(* CODESYS project almacen.project
   Version: 0.0.0.0
   Title: prueba_v2
   Author: Sara

Project tree, tasks and I/O mapping:
  MyController : TM241CE24R, Schneider Electric, order no. TM241CE24R, version 5.0.8.2
    application Application
      libraries: VisuElemBase, * (System); VisuDialogs, * (System)
      task MAST (cyclic, interval 10 ms, priority 15, watchdog 100 ms x 1) calls Main
      task VISU_TASK (cyclic, interval 100 ms, priority 31) calls VisuElems.Visu_Prg
      global variables GVL
      program Main [ST]
      program RecogidaPieza [ST]: Inicio_PiezaEntrada, PiezaDetectada
      program PosicionRobot [ST]
      program TrasladoPieza [ST]: Inicio_TrasladoPieza
      program ExtraerPieza [ST]: Inicio_ExtraerPieza
      program SalidaPieza [ST]: Inicio_SalidaPieza
      program Seguridad [ST]
      program MovimientoRobot [ST]: Inicio_MovimientoRobot, Fin_MovRobot
      program Funcionamiento [ST]: Carga, Descarga, NoAlmacena, CargaDescarga, CD_NoCarga, CD_Carga, CD_Descarga, CD_NoDescarga, ConfirmaCarga
      program Mando [ST]: Inicializar, Automatico, Manual, ParadaSolicitada
      program Acciones [ST]
      program Inicializacion [ST]
      program GestionPiezas [ST]
      program MarchaVSO [ST]: Recoger, Trasladar, Extraer, Salir, Finalizar
      program Comunicacion [CFC]
      program EntradasSalidas [ST]
      text list Pantallas_Lista
      program Control [ST]
      text list Funcionamiento_Lista
      text list Descarga_Lista
      text list DescargaColor_Lista
      program Test [ST]: Subir, Bajar, Estirar, Recoger, Abrir, Cerrar
      text list Test_Lista
      text list Carga_Lista
      Etapas/
        data type Etapas_RecogidaPieza
        data type Etapas_TrasladoPieza
        data type Etapas_ExtraerPieza
        data type Etapas_SalidaPieza
        data type Etapas_Seguridad
        data type Etapas_MovimientoRobot
        data type Etapas_Funcionamiento
        data type Etapas_Mando
        data type Etapas_Inicializacion
        data type Etapas_MarchaVSO
        data type Etapas_Test
      visualisation Pantalla
    DI : Digital Inputs, Schneider Electric, version 5.0.8.2
        input  iwDI_IW0 : WORD  // IW0
        input  ibDI_IB1 : BYTE  // IB1
    DQ : Digital Outputs, Schneider Electric, version 5.0.8.2
        output qwDQ_QW0 : WORD  // QW0
        output qbDQ_QB1 : BYTE  // QB1
    Counters : Counters, Schneider Electric, version 5.0.8.2
    Pulse_Generators : Pulse Generators, Schneider Electric, version 5.0.8.2
    Cartridge_1 : Cartridge, Schneider Electric, version 5.0.8.2
    IO_Bus : IO bus - TM3, Schneider Electric, version 5.0.8.2
    COM_Bus : COM bus, Schneider Electric, version 5.0.8.2
    Ethernet_1 : Ethernet Network, Schneider Electric, version 5.0.8.2
        settings: IPAddress = [10, 11, 164, 211]; SubnetMask = [255, 255, 252, 0]; WebServer = TRUE; FTP Server = TRUE; SoMachine Protocol = TRUE; Modbus Server = TRUE; NetManage Protocol = TRUE; SNMP protocol = TRUE; Enable Routing = FALSE; WebVisu protocol = TRUE; DHCP Server Active = TRUE
    Serial_Line_1 : Serial line, Schneider Electric, version 5.0.8.2
      Machine_Expert_Network_Manager : Machine Expert-Network Manager, Schneider Electric, version 4.0.0.3
    Serial_Line_2 : Serial line, Schneider Electric, version 5.0.8.2
      Modbus_Manager : Modbus Manager, Schneider Electric, version 4.0.0.3
  libraries: VisuSymbols, 3.5.10.0 (System)
  text list GlobalTextList
*)

// MyController/Application/Etapas/Etapas_RecogidaPieza
{attribute 'qualified_only'}
{attribute 'strict'}
TYPE Etapas_RecogidaPieza :
(
	EInicial, RecogerCilindro1, MoverRobot, AccionarCilindro, DetectarPieza,
	Espera, BajarRobot, CerrarPinza, SubirRobot, RecogerCilindro2 
);
END_TYPE

// MyController/Application/Etapas/Etapas_TrasladoPieza
{attribute 'qualified_only'}
{attribute 'strict'}
TYPE Etapas_TrasladoPieza :
(
	EInicial, MoverRobot, AccionarCilindro, BajarRobot, AbrirPinza, SubirRobot, 
	RecogerCilindro, Fin
);
END_TYPE

// MyController/Application/Etapas/Etapas_ExtraerPieza
{attribute 'qualified_only'}
{attribute 'strict'}
TYPE Etapas_ExtraerPieza :
(
	EInicial, RecogerCilindro1, MoverRobot, AccionarCilindro, BajarRobot, CerrarPinza,
	SubirRobot, RecogerCilindro2, Espera
);
END_TYPE

// MyController/Application/Etapas/Etapas_SalidaPieza
{attribute 'qualified_only'}
{attribute 'strict'}
TYPE Etapas_SalidaPieza :
(
	EInicial, MoverRobot, AccionarCilindro, AbrirPinza, SubirRobot, RecogerCilindro, Fin
);
END_TYPE

// MyController/Application/Etapas/Etapas_Seguridad
{attribute 'qualified_only'}
{attribute 'strict'}
TYPE Etapas_Seguridad :
(
	Normal, D1, Rearme
);
END_TYPE

// MyController/Application/Etapas/Etapas_MovimientoRobot
{attribute 'qualified_only'}
{attribute 'strict'}
TYPE Etapas_MovimientoRobot :
(
	EInicial, EnvioVertical, MovVertical, EnvioHorizontal, MovHorizontal, Fin
);
END_TYPE

// MyController/Application/Etapas/Etapas_Funcionamiento
{attribute 'qualified_only'}
{attribute 'strict'}
TYPE Etapas_Funcionamiento :
(
	EInicial, Modo, RecogePieza1, SalidaPieza, RecogePieza2, TrasladoPieza, Espera,
	ExtraePieza, EsperaCD_Carga, EsperaCD_Descarga, SalidaPieza2, Fin
);
END_TYPE

// MyController/Application/Etapas/Etapas_Mando
{attribute 'qualified_only'}
{attribute 'strict'}
TYPE Etapas_Mando :
(
	A1, A2, A6, F1, F4, F6
);
END_TYPE

// MyController/Application/Etapas/Etapas_Inicializacion
{attribute 'qualified_only'}
{attribute 'strict'}
TYPE Etapas_Inicializacion :
(
	EInicial, Espera, MoverRobot, Fin
);
END_TYPE

// MyController/Application/Etapas/Etapas_MarchaVSO
{attribute 'qualified_only'}
{attribute 'strict'}
TYPE Etapas_MarchaVSO :
(
	EInicial, Funcionamiento, RecogePieza, TrasladoPieza, ExtraePieza, SalidaPieza, Espera, Fin
);
END_TYPE

// MyController/Application/Etapas/Etapas_Test
{attribute 'qualified_only'}
{attribute 'strict'}
TYPE Etapas_Test :
(
	EInicial, Espera, Funcionamiento, MoverRobot, SubirRobot, BajarRobot, AccionarCilindro, RecogerCilindro,
	AbrirPinza, CerrarPinza, Fin
);
END_TYPE

// MyController/Application/GVL
{attribute 'qualified_only'}
VAR_GLOBAL
	// Selector (AUTO=0, MAN=1)
	IN_Aut_Man: BOOL;
	// Final de carrera activado con el cilindro recogido
	IN_FC_CilindroAtras: BOOL;
	// Final de carrera activado con el cilindro accionado
	IN_FC_CilindroDelante: BOOL;
	// Final del movimiento horizontal del robot detectado
	IN_Fin_EjeHorizontal: BOOL;
	// Final del movimiento vertical del robot detectado
	IN_Fin_EjeVertical: BOOL;
	// Detector de pieza negra
	IN_PiezaNegra: BOOL;
	// Detector de pieza roja
	IN_PiezaRoja: BOOL;
	// Detector de pieza plateada
	IN_PiezaPlateada: BOOL;
	// Pulsador Reset
	IN_Reset: BOOL;
	// Seta de emergencia
	IN_Seta_Emergencia: BOOL;
	// Pulsador Start
	IN_Start: BOOL;
	// Pulsador Stop
	IN_Stop: BOOL;
	// Bit de posición 0
	OUT_Bit_Posicion0: BOOL;
	// Bit de posición 1
	OUT_Bit_Posicion1: BOOL;
	// Bit de posición 2
	OUT_Bit_Posicion2: BOOL;
	// Accionar el cilindro
	OUT_Cilindro: BOOL;
	// Inicio del movimiento horizontal del robot
	OUT_EjeHorizontal: BOOL;
	// Inicio del movimiento vertical del robot
	OUT_EjeVertical: BOOL;
	// Piloto Q1
	OUT_Piloto_Q1: BOOL;
	// Piloto Q2
	OUT_Piloto_Q2: BOOL;
	// Piloto Reset
	OUT_Piloto_Reset: BOOL;
	// Piloto Start
	OUT_Piloto_Start: BOOL;
	// Accionar la pinza
	OUT_Pinza: BOOL;
	// Bit que indica que hay una pieza en la entrada 
	// (escrito por la estación de procesado)
	BIT_PiezaEntrada: BOOL;
	// Bit que indica que se ha recogido la pieza de la entrada
	// (leído por la estación de procesado)
	BIT_PiezaRecogida: BOOL;
END_VAR

// MyController/Application/Main
PROGRAM Main
VAR
	VSO_Recoger: BOOL;
	VSO_Extraer: BOOL;
	VSO_Salir: BOOL;
	VSO_Trasladar: BOOL;
	VSO_Nada: BOOL;
	VSO_ColorDescarga: INT;
END_VAR

Comunicacion();
EntradasSalidas();
Funcionamiento();
Mando();
Seguridad();
RecogidaPieza();
TrasladoPieza();
ExtraerPieza();
SalidaPieza();
Inicializacion();
Acciones();
MovimientoRobot();
PosicionRobot();
GestionPiezas();
MarchaVSO();
Control();
Test();

END_PROGRAM

// MyController/Application/Comunicacion
PROGRAM Comunicacion
VAR
	FB_ADDM: ADDM;
	FB_READ_VAR: READ_VAR;
	FB_WRITE_VAR: WRITE_VAR;
	DataRead: ARRAY [0..0] OF WORD;
	DataWrite: ARRAY [0..0] OF WORD;
	Direccion: ADDRESS;
	addm_exe: BOOL;
	Q_TIMER0:BOOL;
	TON_0: TON;
	CTU0: CTU;
	SR: SR;
END_VAR

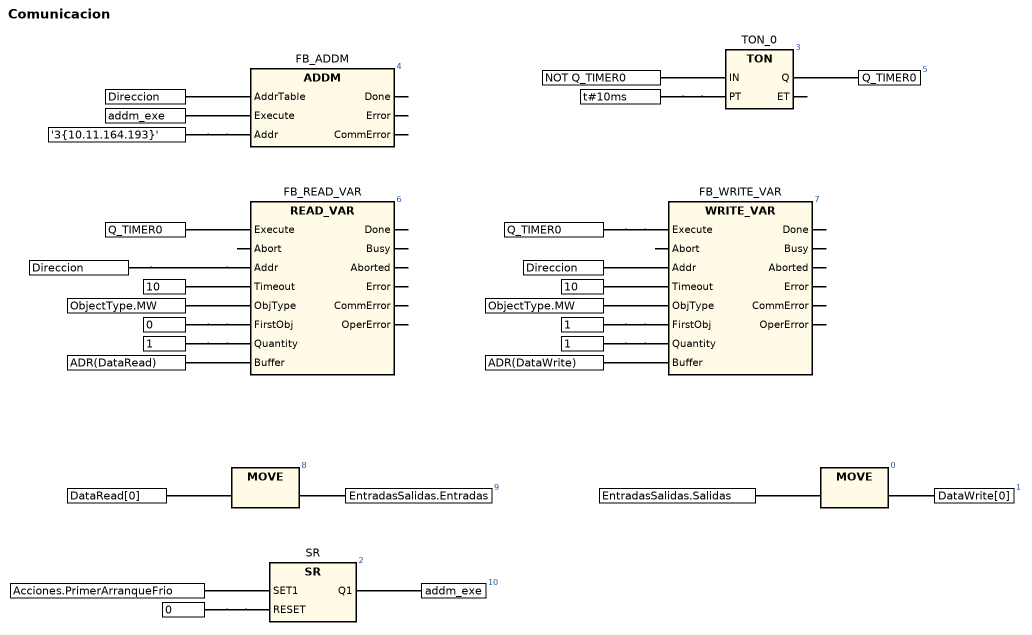
DataWrite[0] := EntradasSalidas.Salidas;
SR(SET1 := Acciones.PrimerArranqueFrio, RESET := 0);
TON_0(IN := NOT Q_TIMER0, PT := t#10ms); // TON
FB_ADDM(AddrTable := Direccion, Execute := addm_exe, Addr := '3{10.11.164.193}'); // ADDM
Q_TIMER0 := TON_0.Q;
FB_READ_VAR(
    Execute := Q_TIMER0,
    Addr := Direccion,
    Timeout := 10,
    ObjType := ObjectType.MW,
    FirstObj := 0,
    Quantity := 1,
    Buffer := ADR(DataRead)); // READ_VAR
FB_WRITE_VAR(
    Execute := Q_TIMER0,
    Addr := Direccion,
    Timeout := 10,
    ObjType := ObjectType.MW,
    FirstObj := 1,
    Quantity := 1,
    Buffer := ADR(DataWrite)); // WRITE_VAR
EntradasSalidas.Entradas := DataRead[0];
addm_exe := SR.Q1;

END_PROGRAM

// MyController/Application/EntradasSalidas
PROGRAM EntradasSalidas
VAR_INPUT
	Entradas: WORD;
END_VAR
VAR
	Salidas: WORD;
END_VAR

(*ENTRADAS*)
GVL.IN_Start := Entradas.0;
GVL.IN_Stop := Entradas.1;
GVL.IN_Reset := Entradas.3;
GVL.IN_Seta_Emergencia := Entradas.5;
GVL.IN_FC_CilindroAtras := Entradas.8;
GVL.IN_FC_CilindroDelante := Entradas.9;
GVL.IN_PiezaNegra := Entradas.10;
GVL.IN_PiezaRoja := Entradas.11;
GVL.IN_PiezaPlateada := Entradas.12;
GVL.IN_Fin_EjeVertical := Entradas.13;
GVL.IN_Fin_EjeHorizontal := Entradas.14;
GVL.BIT_PiezaEntrada := Entradas.15;

(*SALIDAS*)
Salidas.0 := GVL.OUT_Piloto_Start;
Salidas.1 := GVL.OUT_Piloto_Reset;
Salidas.2 := GVL.OUT_Piloto_Q1;
Salidas.3 := GVL.OUT_Piloto_Q2;
Salidas.4 := GVL.OUT_Cilindro;
Salidas.5 := GVL.OUT_Pinza;
Salidas.6 := GVL.OUT_Bit_Posicion0;
Salidas.7 := GVL.OUT_Bit_Posicion1;
Salidas.8 := GVL.OUT_Bit_Posicion2;
Salidas.9 := GVL.OUT_EjeVertical;
Salidas.10 := GVL.OUT_EjeHorizontal;
Salidas.11 := GVL.BIT_PiezaRecogida;

END_PROGRAM

// MyController/Application/Acciones
PROGRAM Acciones
VAR
	SET_Cilindro: BOOL;
	RESET_Cilindro: BOOL;
	SET_Pinza: BOOL;
	RESET_Pinza: BOOL;
	BLINK: BLINK;
	PrimerArranqueFrio: BOOL;
	SR_1: SR;
	SR_3: SR;
	SR_4: SR;
	Parpadeo: BOOL;
	TON: ton;
	Tiempo_350ms: BOOL;
	EntradaTON350ms: BOOL;
	TON_3: TON;
	EntradaTON500ms: BOOL;
	Tiempo_500ms: BOOL;
	TON_2: TON;
	EntradaTON1s: BOOL;
	Tiempo_1s: BOOL;
END_VAR

(*PARADA DE EMERGENCIA*)
IF Seguridad.Estado = Etapas_Seguridad.D1 THEN
	RecogidaPieza.Estado := Etapas_RecogidaPieza.EInicial;
	TrasladoPieza.Estado := Etapas_TrasladoPieza.EInicial;
	ExtraerPieza.Estado := Etapas_ExtraerPieza.EInicial;
	SalidaPieza.Estado := Etapas_SalidaPieza.EInicial;
	MovimientoRobot.Estado := Etapas_MovimientoRobot.EInicial;
	Mando.Estado := Etapas_Mando.A1;
	Funcionamiento.Estado := Etapas_Funcionamiento.EInicial;
	Inicializacion.Estado := Etapas_Inicializacion.EInicial;
	MarchaVSO.Estado := Etapas_MarchaVSO.EInicial;
END_IF

(*REARME*)
IF Seguridad.Estado = Etapas_Seguridad.Rearme THEN
	Mando.Estado := Etapas_Mando.A6;
END_IF


(*GUARDAR FECHA Y COLOR TEMPORAL PARA LA GESTIÓN DE PIEZAS*)
IF RecogidaPieza.Estado = Etapas_RecogidaPieza.DetectarPieza THEN
	IF GVL.IN_PiezaNegra THEN
		RecogidaPieza.ColorPieza := 1;
		RecogidaPieza.Fecha := getRTC();
	ELSIF GVL.IN_PiezaPlateada THEN
		RecogidaPieza.ColorPieza := 2;
		RecogidaPieza.Fecha := getRTC();
	ELSIF GVL.IN_PiezaRoja THEN
		RecogidaPieza.ColorPieza := 3;
		RecogidaPieza.Fecha := getRTC();
	END_IF 
END_IF


(*ACCIONAMIENTO DEL CILINDRO*)
IF RecogidaPieza.Estado = Etapas_RecogidaPieza.AccionarCilindro OR TrasladoPieza.Estado = Etapas_TrasladoPieza.AccionarCilindro OR 
	ExtraerPieza.Estado = Etapas_ExtraerPieza.AccionarCilindro OR SalidaPieza.Estado = Etapas_SalidaPieza.AccionarCilindro OR
	Test.Estado = Etapas_Test.AccionarCilindro THEN
	  SET_Cilindro := 1;
ELSE			
	  SET_Cilindro := 0;	
END_IF

(*RECOGIDA DEL CILINDRO*)
IF RecogidaPieza.Estado = Etapas_RecogidaPieza.RecogerCilindro1 OR RecogidaPieza.Estado = Etapas_RecogidaPieza.RecogerCilindro2 OR
	TrasladoPieza.Estado = Etapas_TrasladoPieza.RecogerCilindro OR ExtraerPieza.Estado = Etapas_ExtraerPieza.RecogerCilindro1 OR
	ExtraerPieza.Estado = Etapas_ExtraerPieza.RecogerCilindro2 OR SalidaPieza.Estado = Etapas_SalidaPieza.RecogerCilindro 
	OR Inicializacion.Estado = Etapas_Inicializacion.Espera OR Seguridad.Estado = Etapas_Seguridad.D1 OR
	Test.Estado = Etapas_Test.RecogerCilindro THEN
	  RESET_Cilindro := 1;
ELSE			
	  RESET_Cilindro := 0;	
END_IF

(*ABRIR LA PINZA*)
IF TrasladoPieza.Estado = Etapas_TrasladoPieza.AbrirPinza OR SalidaPieza.Estado = Etapas_SalidaPieza.AbrirPinza OR
	Inicializacion.Estado = Etapas_Inicializacion.Espera OR Seguridad.Estado = Etapas_Seguridad.D1 OR 
	Test.Estado = Etapas_Test.AbrirPinza THEN
	  RESET_Pinza := 1;
ELSE			
	  RESET_Pinza := 0;	
END_IF

(*CERRAR LA PINZA*)
IF RecogidaPieza.Estado = Etapas_RecogidaPieza.CerrarPinza OR  ExtraerPieza.Estado = Etapas_ExtraerPieza.CerrarPinza OR
	Test.Estado = Etapas_Test.CerrarPinza THEN
	  SET_Pinza:= 1;
ELSE			
	  SET_Pinza := 0;	
END_IF


(*ARRANQUE FRÍO*)
PrimerArranqueFrio := IsFirstMastColdCycle();
SR_1(SET1:= PrimerArranqueFrio, RESET:= Mando.Estado = Etapas_Mando.A6, Q1=> Mando.ArranqueFrio);


(*TEMPORIZADOR 350ms*)
IF MovimientoRobot.Estado = Etapas_MovimientoRobot.EnvioVertical OR MovimientoRobot.Estado = Etapas_MovimientoRobot.EnvioHorizontal  THEN
		EntradaTON350ms := 1;
ELSE
		EntradaTON350ms := 0;
END_IF
TON(IN:= EntradaTON350ms, PT:= T#350MS, Q=> Tiempo_350ms);

(*TEMPORIZADOR 1s*)
IF TrasladoPieza.Estado = Etapas_TrasladoPieza.MoverRobot THEN
	EntradaTON1s := 1;
ELSE
	EntradaTON1s := 0;
END_IF
TON_2(IN:= EntradaTON1s, PT:= T#1S, Q=> Tiempo_1s);

(*TEMPORIZADOR 500ms*)
IF RecogidaPieza.Estado = Etapas_RecogidaPieza.DetectarPieza  OR MovimientoRobot.Estado = Etapas_MovimientoRobot.MovVertical OR 
	MovimientoRobot.Estado = Etapas_MovimientoRobot.MovHorizontal OR RecogidaPieza.Estado = Etapas_RecogidaPieza.Espera THEN
	EntradaTON500ms := 1;
ELSE
	EntradaTON500ms := 0;
END_IF
TON_3(IN:= EntradaTON500ms, PT:= T#500MS, Q=> Tiempo_500ms);

BLINK(ENABLE:= TRUE, TIMELOW:= T#500MS, TIMEHIGH:= T#500MS, OUT=> Parpadeo);


(*SALIDAS*)
(*BIT_PIEZARECOGIDA*)
GVL.BIT_PiezaRecogida := RecogidaPieza.Estado = Etapas_RecogidaPieza.Espera;

(*OUT_CILINDRO*)
SR_3(SET1:= SET_Cilindro , RESET:= RESET_Cilindro, Q1=> GVL.OUT_Cilindro );

(*OUT_PINZA*)
SR_4(SET1:= SET_Pinza , RESET:= RESET_Pinza, Q1=> GVL.OUT_Pinza );

(*OUT_BIT_POSICION*)
CASE PosicionRobot.EnviarCoordenadas OF
	0: GVL.OUT_Bit_Posicion2:=0; GVL.OUT_Bit_Posicion1:=0; GVL.OUT_Bit_Posicion0:=0;
	1: GVL.OUT_Bit_Posicion2:=0; GVL.OUT_Bit_Posicion1:=0; GVL.OUT_Bit_Posicion0:=1;
	2: GVL.OUT_Bit_Posicion2:=0; GVL.OUT_Bit_Posicion1:=1; GVL.OUT_Bit_Posicion0:=0;
	3: GVL.OUT_Bit_Posicion2:=0; GVL.OUT_Bit_Posicion1:=1; GVL.OUT_Bit_Posicion0:=1;
	4: GVL.OUT_Bit_Posicion2:=1; GVL.OUT_Bit_Posicion1:=0; GVL.OUT_Bit_Posicion0:=0;
	5: GVL.OUT_Bit_Posicion2:=1; GVL.OUT_Bit_Posicion1:=0; GVL.OUT_Bit_Posicion0:=1;
	6: GVL.OUT_Bit_Posicion2:=1; GVL.OUT_Bit_Posicion1:=1; GVL.OUT_Bit_Posicion0:=0;
	7: GVL.OUT_Bit_Posicion2:=1; GVL.OUT_Bit_Posicion1:=1; GVL.OUT_Bit_Posicion0:=1;
END_CASE

(*OUT_EJEVERTICAL*)
IF MovimientoRobot.Estado = Etapas_MovimientoRobot.MovVertical THEN
	GVL.OUT_EjeVertical := 1;
ELSE 
	GVL.OUT_EjeVertical := 0;
END_IF

(*OUT_EJEHORIZONTAL*)
IF MovimientoRobot.Estado = Etapas_MovimientoRobot.MovHorizontal THEN
	GVL.OUT_EjeHorizontal := 1;
ELSE
	GVL.OUT_EjeHorizontal := 0;
END_IF

(*OUT_PILOTO_Q1*)
(*Se enciende de forma continua cuando la estación está EN FUNCIONAMIENTO, parpadea cuando ESTÁ PARADA*)
GVL.OUT_Piloto_Q1 := (Mando.Estado = Etapas_Mando.F1 OR Mando.Estado = Etapas_Mando.F4 OR Mando.Estado = Etapas_Mando.F6 OR Mando.Estado = Etapas_Mando.A2) OR 
					(Mando.Estado = Etapas_Mando.A1 AND Parpadeo);
						
(*OUT_PILOTO_Q2*)
(*Se enciende de forma continua cuando la estación puede recibir una pieza, parpadea cuando el almacén está lleno*)
GVL.OUT_Piloto_Q2 := ((Mando.Estado = Etapas_Mando.F1 OR Mando.Estado = Etapas_Mando.A2 OR Mando.Estado = Etapas_Mando.F6 OR Mando.Estado = Etapas_Mando.F4
					OR Mando.Estado = Etapas_Mando.A1) AND GestionPiezas.ContadorTotal<18) OR (GestionPiezas.ContadorTotal=18 AND Parpadeo);
					
(*OUT_PILOTO_RESET*)
(*Se enciende de forma continua cuando la estación se está inicializando, parpadea para pulsar RESET*)
GVL.OUT_Piloto_Reset := (Mando.Estado = Etapas_Mando.A6 AND Inicializacion.Estado = Etapas_Inicializacion.MoverRobot) 
						OR (Mando.Estado = Etapas_Mando.A6 AND Inicializacion.Estado = Etapas_Inicializacion.Espera AND Parpadeo);

(*OUT_PILOTO_START*)
(*Se enciende de forma continua cuando HAY UNA PETICIÓN DE PARO, parpadea para pulsar START*)
GVL.OUT_Piloto_Start := (Mando.Estado = Etapas_Mando.F4 OR Mando.Estado = Etapas_Mando.A2) OR ((Mando.Estado = Etapas_Mando.A1 OR
						 Test.Estado = Etapas_Test.Funcionamiento OR Test.Estado = Etapas_Test.Espera) AND Parpadeo);

END_PROGRAM

// MyController/Application/Seguridad
PROGRAM Seguridad
VAR_INPUT
	Estado: Etapas_Seguridad;
END_VAR

(*MÁQUINA DE ESTADOS SEGURIDAD*)

CASE Estado OF
	
	Etapas_Seguridad.Normal:
	(*Transición*)
	IF NOT GVL.IN_Seta_Emergencia THEN
		Estado := Etapas_Seguridad.D1;
	END_IF
	
	Etapas_Seguridad.D1:
	(*Parada de emergencia, pone las máquinas de estado en la etapa inicial*)
	(*Transición*)
	IF GVL.IN_Seta_Emergencia THEN
		Estado := Etapas_Seguridad.Rearme;
	END_IF
	
	Etapas_Seguridad.Rearme:
	(*Salta a la etapa A6 de inicialización*)
		Estado := Etapas_Seguridad.Normal;		

END_CASE

END_PROGRAM

// MyController/Application/RecogidaPieza
PROGRAM RecogidaPieza
VAR_INPUT
	Estado: Etapas_RecogidaPieza;
	ColorPieza: INT;
	Fecha: DINT;
END_VAR

(*MÁQUINA DE ESTADOS PARA RECOGER LA PIEZA EN LA ENTRADA*)

CASE Estado OF
	
	Etapas_RecogidaPieza.EInicial:
	(*Transición*)
	IF Inicio_PiezaEntrada THEN
		Estado := Etapas_RecogidaPieza.RecogerCilindro1;
	END_IF
	
	Etapas_RecogidaPieza.RecogerCilindro1:
	(*Recoger el cilindro*)
	(*Transición*)
	IF GVL.IN_FC_CilindroAtras THEN
		Estado := Etapas_RecogidaPieza.MoverRobot;
	END_IF
	
	Etapas_RecogidaPieza.MoverRobot:
	(*Mover robot a la posición de entrada*)
	(*Transición*)
	IF MovimientoRobot.Estado = Etapas_MovimientoRobot.Fin THEN
		Estado := Etapas_RecogidaPieza.AccionarCilindro;
	END_IF
	
	Etapas_RecogidaPieza.AccionarCilindro:
	(*Accionar el cilindro*)
	(*Transición*)
	IF GVL.IN_FC_CilindroDelante THEN
		Estado := Etapas_RecogidaPieza.DetectarPieza;
	END_IF
	
	Etapas_RecogidaPieza.DetectarPieza:
	(*Detectar pieza en la entrada*)
	(*Transición*)
	IF PiezaDetectada AND Acciones.Tiempo_500ms THEN
		Estado := Etapas_RecogidaPieza.BajarRobot;
	END_IF
			
	Etapas_RecogidaPieza.BajarRobot:
	(*Bajar el robot una posición*)
	(*Transición*)
	IF MovimientoRobot.Estado = Etapas_MovimientoRobot.Fin THEN
		Estado := Etapas_RecogidaPieza.CerrarPinza;
	END_IF	
	
	Etapas_RecogidaPieza.CerrarPinza:
	(*Cerrar la pinza*)
		Estado := Etapas_RecogidaPieza.SubirRobot;
	
	Etapas_RecogidaPieza.SubirRobot:
	(*Subir robot una posición*)
	(*Transición*)
	IF MovimientoRobot.Estado = Etapas_MovimientoRobot.Fin THEN
		Estado := Etapas_RecogidaPieza.RecogerCilindro2;
	END_IF
	
	Etapas_RecogidaPieza.RecogerCilindro2:
	(*Recoger el cilindro*)
	(*Transición*)
	IF GVL.IN_FC_CilindroAtras THEN
		Estado := Etapas_RecogidaPieza.Espera;
	END_IF
	
	Etapas_RecogidaPieza.Espera:
	(*Final de la recogida, espera para el traslado al almacén o a la salida*)
	(*Transición*)
	IF Acciones.Tiempo_500ms THEN
		Estado := Etapas_RecogidaPieza.EInicial;
	END_IF
	
END_CASE

TRANSITION Inicio_PiezaEntrada:
IF Funcionamiento.Estado = Etapas_Funcionamiento.RecogePieza1 OR Funcionamiento.Estado = Etapas_Funcionamiento.RecogePieza2 
 OR MarchaVSO.Estado = Etapas_MarchaVSO.RecogePieza THEN
	Inicio_PiezaEntrada := 1;
ELSE
	Inicio_PiezaEntrada := 0;
END_IF
END_TRANSITION

TRANSITION PiezaDetectada:
PiezaDetectada := GVL.IN_PiezaNegra OR GVL.IN_PiezaPlateada OR GVL.IN_PiezaRoja;
END_TRANSITION

END_PROGRAM

// MyController/Application/MovimientoRobot
PROGRAM MovimientoRobot
VAR_INPUT
	Estado: Etapas_MovimientoRobot;
END_VAR

(*MÁQUINA DE ESTADOS PARA MOVER EL ROBOT*)

CASE Estado OF
	
	Etapas_MovimientoRobot.EInicial:
	(*Transición*)
	IF Inicio_MovimientoRobot THEN
		Estado := Etapas_MovimientoRobot.EnvioHorizontal;
	END_IF
	
	
	Etapas_MovimientoRobot.EnvioHorizontal:
	(*Envío de la coordenada horizontal*)
	IF Acciones.Tiempo_350ms THEN
		Estado := Etapas_MovimientoRobot.MovHorizontal;
	END_IF
		
	Etapas_MovimientoRobot.MovHorizontal:
	(*Movimiento horizontal del robot*)
	(*Transición*)
	IF Acciones.Tiempo_500ms  THEN
		Estado := Etapas_MovimientoRobot.EnvioVertical;
	END_IF		
	
	Etapas_MovimientoRobot.EnvioVertical:
	(*Envío de la coordenada vertical*)
	IF Acciones.Tiempo_350ms THEN
		Estado := Etapas_MovimientoRobot.MovVertical;
	END_IF
	
	Etapas_MovimientoRobot.MovVertical:
	(*Movimiento vertical del robot*)
	(*Transición*)
	IF Fin_MovRobot AND Acciones.Tiempo_500ms THEN
		Estado := Etapas_MovimientoRobot.Fin;
	END_IF
	
	Etapas_MovimientoRobot.Fin:
	(*Final del movimiento del robot*)
		Estado := Etapas_MovimientoRobot.EInicial;

END_CASE

TRANSITION Inicio_MovimientoRobot:
IF RecogidaPieza.Estado = Etapas_RecogidaPieza.BajarRobot OR RecogidaPieza.Estado = Etapas_RecogidaPieza.MoverRobot OR
	RecogidaPieza.Estado = Etapas_RecogidaPieza.SubirRobot THEN
	
		Inicio_MovimientoRobot := 1;
		
ELSIF TrasladoPieza.Estado = Etapas_TrasladoPieza.MoverRobot OR TrasladoPieza.Estado = Etapas_TrasladoPieza.BajarRobot
	OR TrasladoPieza.Estado = Etapas_TrasladoPieza.SubirRobot THEN
	
		Inicio_MovimientoRobot := 1;
		
ELSIF ExtraerPieza.Estado = Etapas_ExtraerPieza.BajarRobot OR ExtraerPieza.Estado = Etapas_ExtraerPieza.MoverRobot OR
	  ExtraerPieza.Estado = Etapas_ExtraerPieza.SubirRobot THEN
	  
	  Inicio_MovimientoRobot := 1;
	  
ELSIF SalidaPieza.Estado = Etapas_SalidaPieza.MoverRobot OR SalidaPieza.Estado = Etapas_SalidaPieza.SubirRobot THEN
	  
	  Inicio_MovimientoRobot := 1;
	  
ELSIF Inicializacion.Estado = Etapas_Inicializacion.MoverRobot THEN
	
	Inicio_MovimientoRobot := 1;

ELSIF Test.Estado = Etapas_Test.MoverRobot OR Test.Estado = Etapas_Test.SubirRobot OR Test.Estado = Etapas_Test.BajarRobot THEN
	
	Inicio_MovimientoRobot := 1;	

ELSE	
	  Inicio_MovimientoRobot := 0;	
END_IF
END_TRANSITION

TRANSITION Fin_MovRobot:
Fin_MovRobot := GVL.IN_Fin_EjeHorizontal AND GVL.IN_Fin_EjeVertical;
END_TRANSITION

END_PROGRAM

// MyController/Application/TrasladoPieza
PROGRAM TrasladoPieza
VAR_INPUT
	Estado: Etapas_TrasladoPieza;
END_VAR

(*MÁQUINA DE ESTADOS PARA EL TRASLADO DE LA PIEZA AL ALMACÉN*)

CASE Estado OF
	
	Etapas_TrasladoPieza.EInicial:
	(*Transición*)
	IF Inicio_TrasladoPieza THEN
		Estado := Etapas_TrasladoPieza.MoverRobot;
	END_IF
	
	Etapas_TrasladoPieza.MoverRobot:
	(*Mover robot a la posición del almacén*)
	(*Transición*)
	IF MovimientoRobot.Estado = Etapas_MovimientoRobot.Fin AND Acciones.Tiempo_1s THEN
		Estado := Etapas_TrasladoPieza.AccionarCilindro;
	END_IF
	
	Etapas_TrasladoPieza.AccionarCilindro:
	(*Accionar el cilindro*)
	(*Transición*)
	IF GVL.IN_FC_CilindroDelante THEN
		Estado := Etapas_TrasladoPieza.BajarRobot;
	END_IF
	
	Etapas_TrasladoPieza.BajarRobot:
	(*Bajar el robot una posición*)
	(*Transición*)
	IF MovimientoRobot.Estado = Etapas_MovimientoRobot.Fin THEN
		Estado := Etapas_TrasladoPieza.AbrirPinza;
	END_IF
	
	Etapas_TrasladoPieza.AbrirPinza:
	(*Abrir la pinza*)	
		Estado := Etapas_TrasladoPieza.SubirRobot;
		
	Etapas_TrasladoPieza.SubirRobot:
	(*Subir el robot una posición*)
	(*Transición*)
	IF MovimientoRobot.Estado = Etapas_MovimientoRobot.Fin THEN
		Estado := Etapas_TrasladoPieza.RecogerCilindro;
	END_IF
	
	Etapas_TrasladoPieza.RecogerCilindro:
	(*Recoger el cilindro*)
	(*Transición*)
	IF GVL.IN_FC_CilindroAtras THEN
		Estado := Etapas_TrasladoPieza.Fin;
	END_IF
	
	Etapas_TrasladoPieza.Fin:
	(*Final del traslado*)
		Estado := Etapas_TrasladoPieza.EInicial;

END_CASE

TRANSITION Inicio_TrasladoPieza:
IF Funcionamiento.Estado = Etapas_Funcionamiento.TrasladoPieza OR MarchaVSO.Estado = Etapas_MarchaVSO.TrasladoPieza THEN
	Inicio_TrasladoPieza := 1;
ELSE
	Inicio_TrasladoPieza := 0;
END_IF
END_TRANSITION

END_PROGRAM

// MyController/Application/Funcionamiento
PROGRAM Funcionamiento
VAR_INPUT
	Estado: Etapas_Funcionamiento;
END_VAR
VAR
	CargaDisponible: BOOL;
	DescargaDisponible: BOOL;
	ModoFuncionamiento: INT;
	ModoDescarga: INT;
	CargaPorColor: INT;
	DescargaColor: INT;
	BorrarLotes: BOOL;
END_VAR
VAR_INPUT
	NegrasPedidas: INT;
	PlateadasPedidas: INT;
	RojasPedidas: INT;
END_VAR

(*MÁQUINA DE ESTADOS DEL FUNCIONAMIENTO AUTOMÁTICO*)

CASE Estado OF
	
	Etapas_Funcionamiento.EInicial:
	(*Transición*)
	IF Mando.Estado = Etapas_Mando.F1 THEN
		Estado := Etapas_Funcionamiento.Modo;
	END_IF	
	
	Etapas_Funcionamiento.Modo:
	(*MODO DE FUNCIONAMIENTO*)
	(*Transiciones*)
	IF Carga THEN
		Estado := Etapas_Funcionamiento.RecogePieza1;
	ELSIF Descarga THEN
		Estado := Etapas_Funcionamiento.ExtraePieza;
	ELSIF NoAlmacena THEN
		Estado := Etapas_Funcionamiento.RecogePieza2;
	ELSIF CargaDescarga THEN
		Estado := Etapas_Funcionamiento.EsperaCD_Carga;
	ELSIF GVL.IN_Aut_Man THEN
		Estado := Etapas_Funcionamiento.Fin;
	END_IF
	
	(*MODO CARGA*)
	Etapas_Funcionamiento.RecogePieza1:
	(*Recoge la pieza en la entrada*)
	(*Transición*)
	IF RecogidaPieza.Estado = Etapas_RecogidaPieza.Espera AND CargaPorColor = 1 THEN
		Estado := Etapas_Funcionamiento.Espera;
	ELSIF RecogidaPieza.Estado = Etapas_RecogidaPieza.Espera AND CargaPorColor = 0 THEN
		Estado := Etapas_Funcionamiento.TrasladoPieza;
	END_IF
	
	Etapas_Funcionamiento.Espera:
	(*Carga la pieza en el almacén dependiendo del color de la pieza recogida y 
	de que las piezas de ese color que haya almacenadas sean menos de 6*)
	(*Transición*)
	IF ConfirmaCarga THEN
		Estado := Etapas_Funcionamiento.TrasladoPieza;
	ELSIF NOT ConfirmaCarga AND ModoFuncionamiento = 1 THEN
		Estado := Etapas_Funcionamiento.SalidaPieza;
	ELSIF NOT ConfirmaCarga AND ModoFuncionamiento = 4 THEN
		Estado := Etapas_Funcionamiento.SalidaPieza2;
	END_IF
	
	Etapas_Funcionamiento.TrasladoPieza:
	(*Traslada la pieza al almacén*)
	(*Transición*)
	IF TrasladoPieza.Estado = Etapas_TrasladoPieza.Fin AND ModoFuncionamiento = 1 THEN
		Estado := Etapas_Funcionamiento.Fin;
	ELSIF TrasladoPieza.Estado = Etapas_TrasladoPieza.Fin AND ModoFuncionamiento = 4 THEN
		Estado := Etapas_Funcionamiento.EsperaCD_Descarga;
	END_IF
	
	
	(*MODO DESCARGA*)
	Etapas_Funcionamiento.ExtraePieza:
	(*Extrae pieza del almacén*)
	(*Transición*)
	IF ExtraerPieza.Estado = Etapas_ExtraerPieza.Espera THEN
		Estado := Etapas_Funcionamiento.SalidaPieza;
	END_IF
	
	
	(*MODO NO ALMACENA*)
	Etapas_Funcionamiento.RecogePieza2:
	(*Recoge pieza en la entrada*)
	(*Transición*)
	IF RecogidaPieza.Estado = Etapas_RecogidaPieza.Espera THEN
		Estado := Etapas_Funcionamiento.SalidaPieza;
	END_IF
	
	
	(*MODO CARGA Y DESCARGA*)	
	Etapas_Funcionamiento.EsperaCD_Carga:
	(*Contempla si el almacén está lleno para poder cargar la pieza*)
	(*Transiciones*)
	IF CD_NoCarga THEN
		Estado := Etapas_Funcionamiento.EsperaCD_Descarga;
	ELSIF CD_Carga THEN
		Estado := Etapas_Funcionamiento.RecogePieza1;
	END_IF
	
	
	Etapas_Funcionamiento.SalidaPieza2:
	(*Traslada la pieza a la salida*)
	(*Transición*)
	IF SalidaPieza.Estado = Etapas_SalidaPieza.Fin THEN
		Estado := Etapas_Funcionamiento.EsperaCD_Descarga;
	END_IF
	
	
	Etapas_Funcionamiento.EsperaCD_Descarga:
	(*Contempla si hay piezas en el almacén para poder descargar y las condiciones de descarga*)
	(*Transiciones*)
	IF CD_NoDescarga THEN
		Estado := Etapas_Funcionamiento.Fin;
	ELSIF CD_Descarga THEN
		Estado := Etapas_Funcionamiento.ExtraePieza;
	END_IF
	
		
	Etapas_Funcionamiento.SalidaPieza:
	(*Traslada la pieza a la salida*)
	(*Transición*)
	IF SalidaPieza.Estado = Etapas_SalidaPieza.Fin THEN
		Estado := Etapas_Funcionamiento.Fin;
	END_IF
	
	(*FINAL DE CICLO*)
	Etapas_Funcionamiento.Fin:
		Estado := Etapas_Funcionamiento.EInicial;

END_CASE

TRANSITION Carga:
Carga := GVL.BIT_PiezaEntrada AND GestionPiezas.ContadorTotal<18 AND ModoFuncionamiento = 1;
(*Tiene en cuenta que haya una pieza en la entrada y que el almacén no esté lleno*)
END_TRANSITION

TRANSITION Descarga:
IF ModoDescarga = 1 AND GestionPiezas.ContadorTotal>0 THEN
	DescargaDisponible := 1;
	(*Descarga todo el almacén*)
ELSIF ModoDescarga = 2 AND ((DescargaColor = 1 AND GestionPiezas.ContadorNegro>0) OR (DescargaColor = 2 AND GestionPiezas.ContadorPlateado>0) OR
      (DescargaColor = 3 AND GestionPiezas.ContadorRojo>0)) THEN
	  
	DescargaDisponible := 1;
	(*Descarga todas las piezas del color seleccionado*)
ELSIF ModoDescarga = 3 AND (NegrasPedidas <= GestionPiezas.ContadorNegro AND PlateadasPedidas <= GestionPiezas.ContadorPlateado AND
      RojasPedidas <= GestionPiezas.ContadorRojo) AND NOT (NegrasPedidas = 0 AND PlateadasPedidas = 0 AND RojasPedidas = 0)  THEN
	  
	DescargaDisponible := 1;
	(*Descarga un lote de piezas de cada color*)
ELSE
	DescargaDisponible := 0;
END_IF


Descarga := ModoFuncionamiento = 2 AND DescargaDisponible;
END_TRANSITION

TRANSITION NoAlmacena:
NoAlmacena := ModoFuncionamiento = 3 AND GVL.BIT_PiezaEntrada;

(*No se pone la condición ContadorTotal = 18 porque podría hacer la descarga en vez de no almacenar*)
END_TRANSITION

TRANSITION CargaDescarga:
CargaDescarga := ModoFuncionamiento = 4;
END_TRANSITION

TRANSITION CD_NoCarga:
CD_NoCarga := NOT GVL.BIT_PiezaEntrada OR GestionPiezas.ContadorTotal = 18;
END_TRANSITION

TRANSITION CD_Carga:
CD_Carga := GVL.BIT_PiezaEntrada AND GestionPiezas.ContadorTotal<18;
END_TRANSITION

TRANSITION CD_Descarga:
IF ModoDescarga = 1 AND GestionPiezas.ContadorTotal>0 THEN
	CD_Descarga := 1;
	(*Descarga todo el almacén*)
ELSIF ModoDescarga = 2 AND ((DescargaColor = 1 AND GestionPiezas.ContadorNegro>0) OR (DescargaColor = 2 AND GestionPiezas.ContadorPlateado>0) OR
      (DescargaColor = 3 AND GestionPiezas.ContadorRojo>0)) THEN
	  
	CD_Descarga := 1;
	(*Descarga todas las piezas del color seleccionado*)
ELSIF ModoDescarga = 3 AND (NegrasPedidas <= GestionPiezas.ContadorNegro AND PlateadasPedidas <= GestionPiezas.ContadorPlateado AND
      RojasPedidas <= GestionPiezas.ContadorRojo) AND NOT (NegrasPedidas = 0 AND PlateadasPedidas = 0 AND RojasPedidas = 0)  THEN
	  
	CD_Descarga := 1;
	(*Descarga un lote de piezas de cada color*)
ELSE
	CD_Descarga := 0;
END_IF
END_TRANSITION

TRANSITION CD_NoDescarga:
CD_NoDescarga := NOT CD_Descarga;
END_TRANSITION

TRANSITION ConfirmaCarga:
IF (RecogidaPieza.ColorPieza = 1 AND GestionPiezas.ContadorNegro < 6) OR (RecogidaPieza.ColorPieza = 2 AND
	GestionPiezas.ContadorPlateado < 6) OR (RecogidaPieza.ColorPieza = 3 AND GestionPiezas.ContadorRojo < 6) THEN
	ConfirmaCarga := 1;
ELSE
	ConfirmaCarga := 0;
END_IF
END_TRANSITION

END_PROGRAM

// MyController/Application/Mando
PROGRAM Mando
VAR_INPUT
	Estado: Etapas_Mando;
	ArranqueFrio: Bool;
END_VAR
VAR
	Test: Bool;
END_VAR

(*MÁQUINA DE ESTADOS MANDO*)

CASE Estado OF
	
	Etapas_Mando.A1:
	(*Parada en el estado inicial*)
	(*Transiciones*)
	IF Automatico THEN
		Estado := Etapas_Mando.F1;
	ELSIF Manual THEN
		Estado := Etapas_Mando.F4;
	ELSIF Inicializar  THEN
		Estado := Etapas_Mando.A6;
	END_IF
	
	Etapas_Mando.F1:
	(*Producción normal*)
	(*Transiciones*)
	IF ParadaSolicitada THEN
		Estado := Etapas_Mando.A2;
	ELSIF Test THEN
		Estado := Etapas_Mando.F6;
	END_IF
	
	Etapas_Mando.F4:
	(*Marcha de verificación sin orden*)
	(*Transición*)
	IF Test THEN
		Estado := Etapas_Mando.F6;
	ELSIF MarchaVSO.Estado = Etapas_MarchaVSO.Fin THEN
		Estado := Etapas_Mando.A6;
	END_IF
	
	Etapas_Mando.A2:
	(*Parada solicitada al final del ciclo*)
	(*Transición*)
	IF Funcionamiento.Estado = Etapas_Funcionamiento.Fin OR 
		Funcionamiento.Estado = Etapas_Funcionamiento.Modo THEN
		Estado := Etapas_Mando.A1;
	END_IF
	
	Etapas_Mando.F6:
	(*Marcha de test*)
	(*Transición*)
	IF NOT Test THEN
		Estado := Etapas_Mando.A1;
	END_IF
		
	Etapas_Mando.A6:
	(*Puesta del sistema en el estado inicial*)
	(*Transición*)
	IF Inicializacion.Estado = Etapas_Inicializacion.Fin THEN
		Estado := Etapas_Mando.A1;
	END_IF	
END_CASE

TRANSITION Inicializar:
Inicializar := ArranqueFrio AND GVL.IN_Seta_Emergencia;
END_TRANSITION

TRANSITION Automatico:
Automatico := NOT GVL.IN_Aut_Man AND NOT ArranqueFrio AND (GVL.IN_Start OR Control.HMI_Start) AND GVL.IN_Seta_Emergencia;
END_TRANSITION

TRANSITION Manual:
Manual := GVL.IN_Aut_Man AND NOT ArranqueFrio AND (GVL.IN_Start OR Control.HMI_Start) AND GVL.IN_Seta_Emergencia;
END_TRANSITION

TRANSITION ParadaSolicitada:
ParadaSolicitada := (NOT GVL.IN_Stop OR Control.HMI_Stop OR GVL.IN_Aut_Man) AND NOT Test;
(*Parada solicitada si se pulsa STOP o se cambia al modo MANUAL y no se activa el bit TEST*)
END_TRANSITION

END_PROGRAM

// MyController/Application/Test
PROGRAM Test
VAR_INPUT
	Estado: Etapas_Test;
END_VAR
VAR
	ModoTest: INT;
END_VAR

(*MÁQUINA DE ESTADOS PRUEBA TEST*)

CASE Estado OF
	
	Etapas_Test.EInicial:
	(*Transición*)
	IF Mando.Estado = Etapas_Mando.F6  THEN
		Estado := Etapas_Test.Espera;
	END_IF
	
	Etapas_Test.Espera:
	(*Se pulsa START para que el robot inicie el movimiento*)
	(*Transición*)
	IF GVL.IN_Start OR Control.HMI_Start THEN
		Estado := Etapas_Test.MoverRobot;
	END_IF
	
	Etapas_Test.MoverRobot:
	(*Se mueve el robot a la posicion de salida*)
	(*Transición*)
	IF MovimientoRobot.Estado = Etapas_MovimientoRobot.Fin THEN
		Estado := Etapas_Test.Funcionamiento;
	END_IF
	
	Etapas_Test.Funcionamiento:
	(*Se puede subir o bajar el robot, estirar o recoger el cilindro, abrir o cerrar la pinza y terminar el test*)
	(*Transiciones*)
	IF Subir THEN
		Estado := Etapas_Test.SubirRobot;
	ELSIF Bajar THEN
		Estado := Etapas_Test.BajarRobot;
	ELSIF Estirar THEN
		Estado := Etapas_Test.AccionarCilindro;
	ELSIF Recoger THEN
		Estado := Etapas_Test.RecogerCilindro;
	ELSIF Abrir THEN
		Estado := Etapas_Test.AbrirPinza;
	ELSIF Cerrar THEN
		Estado := Etapas_Test.CerrarPinza;
	ELSIF NOT Mando.Test THEN
		Estado := Etapas_Test.Fin;
	END_IF
	
	Etapas_Test.SubirRobot:
	(*Sube el robot a la posición de referencia*)
	(*Transición*)
	IF MovimientoRobot.Estado = Etapas_MovimientoRobot.Fin THEN
		Estado := Etapas_Test.Funcionamiento;
	END_IF
	
	Etapas_Test.BajarRobot:
	(*Baja el robot a la posición de salida*)
	(*Transición*)
	IF MovimientoRobot.Estado = Etapas_MovimientoRobot.Fin THEN
		Estado := Etapas_Test.Funcionamiento;
	END_IF
	
	Etapas_Test.AccionarCilindro:
	(*Accionar el cilindro*)
	(*Transición*)
	IF GVL.IN_FC_CilindroDelante THEN
		Estado := Etapas_Test.Funcionamiento;
	END_IF
	
	Etapas_Test.RecogerCilindro:
	(*Recoger el cilindro*)
	(*Transición*)
	IF GVL.IN_FC_CilindroAtras THEN
		Estado := Etapas_Test.Funcionamiento;
	END_IF
	
	Etapas_Test.AbrirPinza:
	(*Abrir la pinza*)
		Estado := Etapas_Test.Funcionamiento;
	
	Etapas_Test.CerrarPinza:
	(*Cerrar la pinza*)
		Estado := Etapas_Test.Funcionamiento;
		
	Etapas_Test.Fin:
	(*Fin de la prueba*)
		Estado := Etapas_Test.EInicial;	
	
END_CASE

TRANSITION Subir:
Subir := ModoTest = 1  AND (GVL.IN_Start OR Control.HMI_Start);
END_TRANSITION

TRANSITION Bajar:
Bajar := ModoTest = 2 AND (GVL.IN_Start OR Control.HMI_Start);
END_TRANSITION

TRANSITION Estirar:
Estirar := ModoTest = 3 AND GVL.IN_FC_CilindroAtras AND (GVL.IN_Start OR Control.HMI_Start);
END_TRANSITION

TRANSITION Recoger:
Recoger := ModoTest = 4 AND GVL.IN_FC_CilindroDelante AND (GVL.IN_Start OR Control.HMI_Start);
END_TRANSITION

TRANSITION Abrir:
Abrir := ModoTest = 5 AND GVL.OUT_Pinza AND (GVL.IN_Start OR Control.HMI_Start);
END_TRANSITION

TRANSITION Cerrar:
Cerrar := ModoTest = 6 AND NOT GVL.OUT_Pinza AND (GVL.IN_Start OR Control.HMI_Start);
END_TRANSITION

END_PROGRAM

// MyController/Application/Control
PROGRAM Control
VAR
	BloqueoCargaColor: BOOL;
	BloqueoLotes: BOOL;
	BloqueoManPinzaCerrada: BOOL;
	BloqueoManPinzaAbierta: BOOL;
	ColorAutomatico: BOOL;
	ColorManual: BOOL;
	HMI_Start: BOOL;
	HMI_Stop: BOOL;
	HMI_Reset: BOOL;
	InvManual: BOOL;
	InvCarga: BOOL;
	InvDescarga: BOOL;
	InvDesColor: BOOL;
	InvDesLotes: BOOL;
	InvTest: BOOL;
	i: INT;
	PiezaNegra1: BOOL := FALSE;
	PiezaPlateadaRoja1: BOOL;
	InvPlateadaRoja1: BOOL := TRUE;
	InvNegra1: BOOL;
	PiezaNegra2: BOOL := FALSE;
	PiezaPlateadaRoja2: BOOL;
	InvPlateadaRoja2: BOOL := TRUE;
	InvNegra2: BOOL;
	PiezaNegra3: BOOL := FALSE;
	PiezaPlateadaRoja3: BOOL;
	InvPlateadaRoja3: BOOL := TRUE;
	InvNegra3: BOOL;
	PiezaNegra4: BOOL := FALSE;
	PiezaPlateadaRoja4: BOOL;
	InvPlateadaRoja4: BOOL := TRUE;
	InvNegra4: BOOL;
	PiezaNegra5: BOOL := FALSE;
	PiezaPlateadaRoja5: BOOL;
	InvPlateadaRoja5: BOOL := TRUE;
	InvNegra5: BOOL;
	PiezaNegra6: BOOL := FALSE;
	PiezaPlateadaRoja6: BOOL;
	InvPlateadaRoja6: BOOL := TRUE;
	InvNegra6: BOOL;
	PiezaNegra7: BOOL := FALSE;
	PiezaPlateadaRoja7: BOOL;
	InvPlateadaRoja7: BOOL := TRUE;
	InvNegra7: BOOL;
	PiezaNegra8: BOOL := FALSE;
	PiezaPlateadaRoja8: BOOL;
	InvPlateadaRoja8: BOOL := TRUE;
	InvNegra8: BOOL;
	PiezaNegra9: BOOL := FALSE;
	PiezaPlateadaRoja9: BOOL;
	InvPlateadaRoja9: BOOL := TRUE;
	InvNegra9: BOOL;
	PiezaNegra10: BOOL := FALSE;
	PiezaPlateadaRoja10: BOOL;
	InvPlateadaRoja10: BOOL := TRUE;
	InvNegra10: BOOL;
	PiezaNegra11: BOOL := FALSE;
	PiezaPlateadaRoja11: BOOL;
	InvPlateadaRoja11: BOOL := TRUE;
	InvNegra11: BOOL;
	PiezaNegra12: BOOL := FALSE;
	PiezaPlateadaRoja12: BOOL;
	InvPlateadaRoja12: BOOL := TRUE;
	InvNegra12: BOOL;
	PiezaNegra13: BOOL := FALSE;
	PiezaPlateadaRoja13: BOOL;
	InvPlateadaRoja13: BOOL := TRUE;
	InvNegra13: BOOL;
	PiezaNegra14: BOOL := FALSE;
	PiezaPlateadaRoja14: BOOL;
	InvPlateadaRoja14: BOOL := TRUE;
	InvNegra14: BOOL;
	PiezaNegra15: BOOL := FALSE;
	PiezaPlateadaRoja15: BOOL;
	InvPlateadaRoja15: BOOL := TRUE;
	InvNegra15: BOOL;
	PiezaNegra16: BOOL := FALSE;
	PiezaPlateadaRoja16: BOOL;
	InvPlateadaRoja16: BOOL := TRUE;
	InvNegra16: BOOL;
	PiezaNegra17: BOOL := FALSE;
	PiezaPlateadaRoja17: BOOL;
	InvPlateadaRoja17: BOOL := TRUE;
	InvNegra17: BOOL;
	PiezaNegra18: BOOL := FALSE;
	PiezaPlateadaRoja18: BOOL;
	InvPlateadaRoja18: BOOL := TRUE;
	InvNegra18: BOOL;
END_VAR

(*PROGRAMACIÓN DE LA PANTALLA*)
(*10.11.164.211:8080/webvisu.htm*)

(*Oculta las opciones del modo manual*)
InvManual := Mando.Estado = Etapas_Mando.F1 OR Mando.Estado = Etapas_Mando.F6 OR Mando.Estado = Etapas_Mando.A1 OR
			Mando.Estado = Etapas_Mando.A6 OR Mando.Estado = Etapas_Mando.A2;
			
(*Cambia el color del indicador del modo automático o manual*)
ColorAutomatico := Mando.Estado = Etapas_Mando.F1;
ColorManual := Mando.Estado = Etapas_Mando.F4;

(*Bloquea los botones del modo manual dependiendo de si la pinza se encuentra abierta o cerrada*)
BloqueoManPinzaCerrada := GVL.OUT_Pinza;
BloqueoManPinzaAbierta := NOT GVL.OUT_Pinza;

(*Oculta las opciones de carga si no se ha seleccionado este modo de funcionamiento*)
IF Funcionamiento.ModoFuncionamiento = 1 OR Funcionamiento.ModoFuncionamiento = 4 OR Mando.Estado = Etapas_Mando.F4 THEN
	InvCarga := 0;
ELSE
	InvCarga := 1;
END_IF

(*Oculta las opciones de descarga si no se ha seleccionado este modo de funcionamiento*)
IF Funcionamiento.ModoFuncionamiento = 2 OR Funcionamiento.ModoFuncionamiento = 4 THEN
	InvDescarga := 0;
ELSE 
	InvDescarga := 1;
END_IF

(*Oculta el modo de descarga que no se haya seleccionado*)
IF Funcionamiento.ModoDescarga = 2 THEN
	InvDesLotes := 1;
	InvDesColor := 0;
ELSIF Funcionamiento.ModoDescarga = 3 THEN
	InvDesLotes := 0;
	InvDesColor := 1;
ELSE
	InvDesColor := 1;
	InvDesLotes := 1;
END_IF

(*Oculta las opciones de las pruebas de test si no se ha pulsado Test*)
InvTest := NOT Mando.Test;

(*Bloquea la opción de cambiar el modo de carga en cuanto haya alguna pieza almacenada*)
IF GestionPiezas.ContadorTotal > 0 THEN
	BloqueoCargaColor := 1;
ELSE
	BloqueoCargaColor := 0;
END_IF

(*Bloquea el botón de borrar los lotes pedidos si no se encuentra en la etapa inicial de Mando,
por ejemplo, permite borrar los lotes si se ha hecho una parada a fin de ciclo*)
IF Mando.Estado = Etapas_Mando.A1 THEN
	BloqueoLotes := 0;
ELSE
	BloqueoLotes := 1;
END_IF

(*Programación de las elipses que simulan las piezas almacenadas*)
IF TrasladoPieza.Estado = Etapas_TrasladoPieza.Fin OR ExtraerPieza.Estado = Etapas_ExtraerPieza.Espera THEN
	FOR i:=0 TO 17 DO
		IF GestionPiezas.PosicionPiezaAlmacenada[i] = 1 THEN
				IF GestionPiezas.ColorPiezaAlmacenada[i] = 1 THEN
					PiezaNegra1 := 1;
					InvNegra1 := 0;
					InvPlateadaRoja1 := 1;
				ELSIF GestionPiezas.ColorPiezaAlmacenada[i] = 2 THEN
					InvNegra1 := 1;
					InvPlateadaRoja1 := 0;
					PiezaPlateadaRoja1 := 0;
				ELSIF GestionPiezas.ColorPiezaAlmacenada[i] = 3 THEN
					InvNegra1 := 1;
					InvPlateadaRoja1 := 0;	
					PiezaPlateadaRoja1 := 1;		
				END_IF
				EXIT;
		ELSE
			PiezaNegra1 := 0;
			InvNegra1 := 0;
			InvPlateadaRoja1 := 1;
		END_IF 
	END_FOR
	
	FOR i:=0 TO 17 DO
		IF (GestionPiezas.PosicionPiezaAlmacenada[i] = 2 AND Funcionamiento.CargaPorColor = 0) OR 
			(GestionPiezas.PosicionPiezaAlmacenada[i] = 7 AND Funcionamiento.CargaPorColor = 1) THEN
				IF GestionPiezas.ColorPiezaAlmacenada[i] = 1 THEN
					PiezaNegra2 := 1;
					InvNegra2 := 0;
					InvPlateadaRoja2 := 1;
				ELSIF GestionPiezas.ColorPiezaAlmacenada[i] = 2 THEN
					InvNegra2 := 1;
					InvPlateadaRoja2 := 0;
					PiezaPlateadaRoja2 := 0;
				ELSIF GestionPiezas.ColorPiezaAlmacenada[i] = 3 THEN
					InvNegra2 := 1;
					InvPlateadaRoja2 := 0;	
					PiezaPlateadaRoja2 := 1;		
				END_IF
				EXIT;
		ELSE
			PiezaNegra2 := 0;
			InvNegra2 := 0;
			InvPlateadaRoja2 := 1;
		END_IF
	END_FOR 
	
	FOR i:=0 TO 17 DO
		IF (GestionPiezas.PosicionPiezaAlmacenada[i] = 3 AND Funcionamiento.CargaPorColor = 0) OR 
			(GestionPiezas.PosicionPiezaAlmacenada[i] = 13 AND Funcionamiento.CargaPorColor = 1) THEN
				IF GestionPiezas.ColorPiezaAlmacenada[i] = 1 THEN
					PiezaNegra3 := 1;
					InvNegra3 := 0;
					InvPlateadaRoja3 := 1;
				ELSIF GestionPiezas.ColorPiezaAlmacenada[i] = 2 THEN
					InvNegra3 := 1;
					InvPlateadaRoja3 := 0;
					PiezaPlateadaRoja3 := 0;
				ELSIF GestionPiezas.ColorPiezaAlmacenada[i] = 3 THEN
					InvNegra3 := 1;
					InvPlateadaRoja3 := 0;
					PiezaPlateadaRoja3 := 1;			
				END_IF
				EXIT;
		ELSE
			PiezaNegra3 := 0;
			InvNegra3 := 0;
			InvPlateadaRoja3 := 1;
		END_IF
	END_FOR
	
	FOR i:=0 TO 17 DO
		IF (GestionPiezas.PosicionPiezaAlmacenada[i] = 4 AND Funcionamiento.CargaPorColor = 0) OR 
			(GestionPiezas.PosicionPiezaAlmacenada[i] = 2 AND Funcionamiento.CargaPorColor = 1) THEN
				IF GestionPiezas.ColorPiezaAlmacenada[i] = 1 THEN
					PiezaNegra4 := 1;
					InvNegra4 := 0;
					InvPlateadaRoja4 := 1;
				ELSIF GestionPiezas.ColorPiezaAlmacenada[i] = 2 THEN
					InvNegra4 := 1;
					InvPlateadaRoja4 := 0;
					PiezaPlateadaRoja4 := 0;
				ELSIF GestionPiezas.ColorPiezaAlmacenada[i] = 3 THEN
					InvNegra4 := 1;
					InvPlateadaRoja4 := 0;	
					PiezaPlateadaRoja4 := 1;		
				END_IF
				EXIT;
		ELSE
			PiezaNegra4 := 0;
			InvNegra4 := 0;
			InvPlateadaRoja4 := 1;
		END_IF
	END_FOR
	
	FOR i:=0 TO 17 DO
		IF (GestionPiezas.PosicionPiezaAlmacenada[i] = 5 AND Funcionamiento.CargaPorColor = 0) OR 
			(GestionPiezas.PosicionPiezaAlmacenada[i] = 8 AND Funcionamiento.CargaPorColor = 1) THEN
				IF GestionPiezas.ColorPiezaAlmacenada[i] = 1 THEN
					PiezaNegra5 := 1;
					InvNegra5 := 0;
					InvPlateadaRoja5 := 1;
				ELSIF GestionPiezas.ColorPiezaAlmacenada[i] = 2 THEN
					InvNegra5 := 1;
					InvPlateadaRoja5 := 0;
					PiezaPlateadaRoja5 := 0;
				ELSIF GestionPiezas.ColorPiezaAlmacenada[i] = 3 THEN
					InvNegra5 := 1;
					InvPlateadaRoja5 := 0;	
					PiezaPlateadaRoja5 := 1;		
				END_IF
				EXIT;
		ELSE
			PiezaNegra5 := 0;
			InvNegra5 := 0;
			InvPlateadaRoja5 := 1;
		END_IF
	END_FOR
	
	FOR i:=0 TO 17 DO
		IF (GestionPiezas.PosicionPiezaAlmacenada[i] = 6 AND Funcionamiento.CargaPorColor = 0) OR 
			(GestionPiezas.PosicionPiezaAlmacenada[i] = 14 AND Funcionamiento.CargaPorColor = 1) THEN
				IF GestionPiezas.ColorPiezaAlmacenada[i] = 1 THEN
					PiezaNegra6 := 1;
					InvNegra6 := 0;
					InvPlateadaRoja6 := 1;
				ELSIF GestionPiezas.ColorPiezaAlmacenada[i] = 2 THEN
					InvNegra6 := 1;
					InvPlateadaRoja6 := 0;
					PiezaPlateadaRoja6 := 0;
				ELSIF GestionPiezas.ColorPiezaAlmacenada[i] = 3 THEN
					InvNegra6 := 1;
					InvPlateadaRoja6 := 0;
					PiezaPlateadaRoja6 := 1;			
				END_IF
				EXIT;
		ELSE
			PiezaNegra6 := 0;
			InvNegra6 := 0;
			InvPlateadaRoja6 := 1;
		END_IF
	END_FOR
	
	FOR i:=0 TO 17 DO
		IF (GestionPiezas.PosicionPiezaAlmacenada[i] = 7 AND Funcionamiento.CargaPorColor = 0) OR 
			(GestionPiezas.PosicionPiezaAlmacenada[i] = 3 AND Funcionamiento.CargaPorColor = 1) THEN
				IF GestionPiezas.ColorPiezaAlmacenada[i] = 1 THEN
					PiezaNegra7 := 1;
					InvNegra7 := 0;
					InvPlateadaRoja7 := 1;
				ELSIF GestionPiezas.ColorPiezaAlmacenada[i] = 2 THEN
					InvNegra7 := 1;
					InvPlateadaRoja7 := 0;
					PiezaPlateadaRoja7 := 0;
				ELSIF GestionPiezas.ColorPiezaAlmacenada[i] = 3 THEN
					InvNegra7 := 1;
					InvPlateadaRoja7 := 0;	
					PiezaPlateadaRoja7 := 1;		
				END_IF
				EXIT;
		ELSE
			PiezaNegra7 := 0;
			InvNegra7 := 0;
			InvPlateadaRoja7 := 1;
		END_IF
	END_FOR
	
	FOR i:=0 TO 17 DO
		IF (GestionPiezas.PosicionPiezaAlmacenada[i] = 8 AND Funcionamiento.CargaPorColor = 0) OR 
			(GestionPiezas.PosicionPiezaAlmacenada[i] = 9 AND Funcionamiento.CargaPorColor = 1) THEN
				IF GestionPiezas.ColorPiezaAlmacenada[i] = 1 THEN
					PiezaNegra8 := 1;
					InvNegra8 := 0;
					InvPlateadaRoja8 := 1;
				ELSIF GestionPiezas.ColorPiezaAlmacenada[i] = 2 THEN
					InvNegra8 := 1;
					InvPlateadaRoja8 := 0;
					PiezaPlateadaRoja8 := 0;
				ELSIF GestionPiezas.ColorPiezaAlmacenada[i] = 3 THEN
					InvNegra8 := 1;
					InvPlateadaRoja8 := 0;	
					PiezaPlateadaRoja8 := 1;		
				END_IF
				EXIT;
		ELSE
			PiezaNegra8 := 0;
			InvNegra8 := 0;
			InvPlateadaRoja8 := 1;
		END_IF
	END_FOR
	
	FOR i:=0 TO 17 DO
		IF (GestionPiezas.PosicionPiezaAlmacenada[i] = 9 AND Funcionamiento.CargaPorColor = 0) OR 
			(GestionPiezas.PosicionPiezaAlmacenada[i] = 15 AND Funcionamiento.CargaPorColor = 1) THEN
				IF GestionPiezas.ColorPiezaAlmacenada[i] = 1 THEN
					PiezaNegra9 := 1;
					InvNegra9 := 0;
					InvPlateadaRoja9 := 1;
				ELSIF GestionPiezas.ColorPiezaAlmacenada[i] = 2 THEN
					InvNegra9 := 1;
					InvPlateadaRoja9 := 0;
					PiezaPlateadaRoja9 := 0;
				ELSIF GestionPiezas.ColorPiezaAlmacenada[i] = 3 THEN
					InvNegra9 := 1;
					InvPlateadaRoja9 := 0;			
					PiezaPlateadaRoja9 := 1;
				END_IF
				EXIT;
		ELSE
			PiezaNegra9 := 0;
			InvNegra9 := 0;
			InvPlateadaRoja9 := 1;
		END_IF
	END_FOR
	
	FOR i:=0 TO 17 DO
		IF (GestionPiezas.PosicionPiezaAlmacenada[i] = 10 AND Funcionamiento.CargaPorColor = 0) OR 
			(GestionPiezas.PosicionPiezaAlmacenada[i] = 4 AND Funcionamiento.CargaPorColor = 1) THEN
				IF GestionPiezas.ColorPiezaAlmacenada[i] = 1 THEN
					PiezaNegra10 := 1;
					InvNegra10 := 0;
					InvPlateadaRoja10 := 1;
				ELSIF GestionPiezas.ColorPiezaAlmacenada[i] = 2 THEN
					InvNegra10 := 1;
					InvPlateadaRoja10 := 0;
					PiezaPlateadaRoja10 := 0;
				ELSIF GestionPiezas.ColorPiezaAlmacenada[i] = 3 THEN
					InvNegra10 := 1;
					InvPlateadaRoja10 := 0;	
					PiezaPlateadaRoja10 := 1;		
				END_IF
				EXIT;
		ELSE
			PiezaNegra10 := 0;
			InvNegra10 := 0;
			InvPlateadaRoja10 := 1;
		END_IF
	END_FOR
	
	FOR i:=0 TO 17 DO
		IF (GestionPiezas.PosicionPiezaAlmacenada[i] = 11 AND Funcionamiento.CargaPorColor = 0) OR 
			(GestionPiezas.PosicionPiezaAlmacenada[i] = 10 AND Funcionamiento.CargaPorColor = 1) THEN
				IF GestionPiezas.ColorPiezaAlmacenada[i] = 1 THEN
					PiezaNegra11 := 1;
					InvNegra11 := 0;
					InvPlateadaRoja11 := 1;
				ELSIF GestionPiezas.ColorPiezaAlmacenada[i] = 2 THEN
					InvNegra11 := 1;
					InvPlateadaRoja11 := 0;
					PiezaPlateadaRoja11 := 0;
				ELSIF GestionPiezas.ColorPiezaAlmacenada[i] = 3 THEN
					InvNegra11 := 1;
					InvPlateadaRoja11 := 0;	
					PiezaPlateadaRoja11 := 1;		
				END_IF
				EXIT;
		ELSE
			PiezaNegra11 := 0;
			InvNegra11 := 0;
			InvPlateadaRoja11 := 1;
		END_IF
	END_FOR
	
	FOR i:=0 TO 17 DO
		IF (GestionPiezas.PosicionPiezaAlmacenada[i] = 12 AND Funcionamiento.CargaPorColor = 0) OR 
			(GestionPiezas.PosicionPiezaAlmacenada[i] = 16 AND Funcionamiento.CargaPorColor = 1) THEN
				IF GestionPiezas.ColorPiezaAlmacenada[i] = 1 THEN
					PiezaNegra12 := 1;
					InvNegra12 := 0;
					InvPlateadaRoja12 := 1;
				ELSIF GestionPiezas.ColorPiezaAlmacenada[i] = 2 THEN
					InvNegra12 := 1;
					InvPlateadaRoja12 := 0;
					PiezaPlateadaRoja12 := 0;
				ELSIF GestionPiezas.ColorPiezaAlmacenada[i] = 3 THEN
					InvNegra12 := 1;
					InvPlateadaRoja12 := 0;		
					PiezaPlateadaRoja12 := 1;	
				END_IF
				EXIT;
		ELSE
			PiezaNegra12 := 0;
			InvNegra12 := 0;
			InvPlateadaRoja12 := 1;
		END_IF
	END_FOR
	
	FOR i:=0 TO 17 DO
		IF (GestionPiezas.PosicionPiezaAlmacenada[i] = 13 AND Funcionamiento.CargaPorColor = 0) OR 
			(GestionPiezas.PosicionPiezaAlmacenada[i] = 5 AND Funcionamiento.CargaPorColor = 1) THEN
				IF GestionPiezas.ColorPiezaAlmacenada[i] = 1 THEN
					PiezaNegra13 := 1;
					InvNegra13 := 0;
					InvPlateadaRoja13 := 1;
				ELSIF GestionPiezas.ColorPiezaAlmacenada[i] = 2 THEN
					InvNegra13 := 1;
					InvPlateadaRoja13 := 0;
					PiezaPlateadaRoja13 := 0;
				ELSIF GestionPiezas.ColorPiezaAlmacenada[i] = 3 THEN
					InvNegra13 := 1;
					InvPlateadaRoja13 := 0;	
					PiezaPlateadaRoja13 := 1;	
				END_IF
				EXIT;
		ELSE
			PiezaNegra13 := 0;
			InvNegra13 := 0;
			InvPlateadaRoja13 := 1;
		END_IF
	END_FOR
	
	FOR i:=0 TO 17 DO
		IF (GestionPiezas.PosicionPiezaAlmacenada[i] = 14 AND Funcionamiento.CargaPorColor = 0) OR 
			(GestionPiezas.PosicionPiezaAlmacenada[i] = 11 AND Funcionamiento.CargaPorColor = 1) THEN
				IF GestionPiezas.ColorPiezaAlmacenada[i] = 1 THEN
					PiezaNegra14 := 1;
					InvNegra14 := 0;
					InvPlateadaRoja14 := 1;
				ELSIF GestionPiezas.ColorPiezaAlmacenada[i] = 2 THEN
					InvNegra14 := 1;
					InvPlateadaRoja14 := 0;
					PiezaPlateadaRoja14 := 0;
				ELSIF GestionPiezas.ColorPiezaAlmacenada[i] = 3 THEN
					InvNegra14 := 1;
					InvPlateadaRoja14 := 0;		
					PiezaPlateadaRoja14 := 1;	
				END_IF
				EXIT;
		ELSE
			PiezaNegra14 := 0;
			InvNegra14 := 0;
			InvPlateadaRoja14 := 1;
		END_IF
	END_FOR
	
	FOR i:=0 TO 17 DO
		IF (GestionPiezas.PosicionPiezaAlmacenada[i] = 15 AND Funcionamiento.CargaPorColor = 0) OR 
			(GestionPiezas.PosicionPiezaAlmacenada[i] = 17 AND Funcionamiento.CargaPorColor = 1) THEN
				IF GestionPiezas.ColorPiezaAlmacenada[i] = 1 THEN
					PiezaNegra15 := 1;
					InvNegra15 := 0;
					InvPlateadaRoja15 := 1;
				ELSIF GestionPiezas.ColorPiezaAlmacenada[i] = 2 THEN
					InvNegra15 := 1;
					InvPlateadaRoja15 := 0;
					PiezaPlateadaRoja15 := 0;
				ELSIF GestionPiezas.ColorPiezaAlmacenada[i] = 3 THEN
					InvNegra15 := 1;
					InvPlateadaRoja15 := 0;	
					PiezaPlateadaRoja15 := 1;		
				END_IF
				EXIT;
		ELSE
			PiezaNegra15 := 0;
			InvNegra15 := 0;
			InvPlateadaRoja15 := 1;
		END_IF
	END_FOR
	
	FOR i:=0 TO 17 DO
		IF (GestionPiezas.PosicionPiezaAlmacenada[i] = 16 AND Funcionamiento.CargaPorColor = 0) OR 
			(GestionPiezas.PosicionPiezaAlmacenada[i] = 6 AND Funcionamiento.CargaPorColor = 1) THEN
				IF GestionPiezas.ColorPiezaAlmacenada[i] = 1 THEN
					PiezaNegra16 := 1;
					InvNegra16 := 0;
					InvPlateadaRoja16 := 1;
				ELSIF GestionPiezas.ColorPiezaAlmacenada[i] = 2 THEN
					InvNegra16 := 1;
					InvPlateadaRoja16 := 0;
					PiezaPlateadaRoja16 := 0;
				ELSIF GestionPiezas.ColorPiezaAlmacenada[i] = 3 THEN
					InvNegra16 := 1;
					InvPlateadaRoja16 := 0;		
					PiezaPlateadaRoja16 := 1;	
				END_IF
				EXIT;
		ELSE
			PiezaNegra16 := 0;
			InvNegra16 := 0;
			InvPlateadaRoja16 := 1;
		END_IF
	END_FOR
	
	FOR i:=0 TO 17 DO
		IF (GestionPiezas.PosicionPiezaAlmacenada[i] = 17 AND Funcionamiento.CargaPorColor = 0) OR 
			(GestionPiezas.PosicionPiezaAlmacenada[i] = 12 AND Funcionamiento.CargaPorColor = 1) THEN
				IF GestionPiezas.ColorPiezaAlmacenada[i] = 1 THEN
					PiezaNegra17 := 1;
					InvNegra17 := 0;
					InvPlateadaRoja17 := 1;
				ELSIF GestionPiezas.ColorPiezaAlmacenada[i] = 2 THEN
					InvNegra17 := 1;
					InvPlateadaRoja17 := 0;
					PiezaPlateadaRoja17 := 0;
				ELSIF GestionPiezas.ColorPiezaAlmacenada[i] = 3 THEN
					InvNegra17 := 1;
					InvPlateadaRoja17 := 0;	
					PiezaPlateadaRoja17 := 1;		
				END_IF
				EXIT;
		ELSE
			PiezaNegra17 := 0;
			InvNegra17 := 0;
			InvPlateadaRoja17 := 1;
		END_IF
	END_FOR
	
	FOR i:=0 TO 17 DO
		IF GestionPiezas.PosicionPiezaAlmacenada[i] = 18 THEN
				IF GestionPiezas.ColorPiezaAlmacenada[i] = 1 THEN
					PiezaNegra18 := 1;
					InvNegra18 := 0;
					InvPlateadaRoja18 := 1;
				ELSIF GestionPiezas.ColorPiezaAlmacenada[i] = 2 THEN
					InvNegra18 := 1;
					InvPlateadaRoja18 := 0;
					PiezaPlateadaRoja18 := 0;
				ELSIF GestionPiezas.ColorPiezaAlmacenada[i] = 3 THEN
					InvNegra18 := 1;
					InvPlateadaRoja18 := 0;		
					PiezaPlateadaRoja18 := 1;	
				END_IF
				EXIT;
		ELSE
			PiezaNegra18 := 0;
			InvNegra18 := 0;
			InvPlateadaRoja18 := 1;
		END_IF
	END_FOR
END_IF

END_PROGRAM

// MyController/Application/GestionPiezas
PROGRAM GestionPiezas
VAR
	i: INT;
	j: INT;
	k: INT;
	m: INT;
	n: INT;
	ContadorRojo: INT := 0;
	ContadorNegro: INT := 0;
	ContadorPlateado: INT := 0;
	ContadorTotal: INT := 0;
	ColorPiezaAlmacenada: ARRAY [0..17] OF INT;
	FechaPiezaAlmacenada: ARRAY [0..17] OF DINT;
	PosicionPiezaAlmacenada: ARRAY [0..17] OF INT;
	ColorPiezaDescargada: ARRAY [0..17] OF INT;
	FechaPiezaDescargada: ARRAY [0..17] OF DINT;
	PosicionDisponible_aux: BOOL;
	PosicionDisponible: INT;
	PosicionDescarga: INT;
	FechaReferencia: DINT;
END_VAR

(*Posición de la pieza a cargar*)
IF TrasladoPieza.Estado = Etapas_TrasladoPieza.MoverRobot THEN 
	IF Mando.Estado = Etapas_Mando.F1 OR Mando.Estado = Etapas_Mando.F6 OR Mando.Estado = Etapas_Mando.A2 OR
		Mando.Estado = Etapas_Mando.F4 THEN
		IF Funcionamiento.CargaPorColor = 1 THEN
			(*Llena el almacén dependiendo del color: Nivel 1 - negro, Nivel 2 - plateado, Nivel 3 - rojo*)
			IF ((RecogidaPieza.ColorPieza = 1 AND ColorPiezaDescargada[k] = 0) OR ColorPiezaDescargada[k] = 1) AND ContadorNegro < 6 THEN
				FOR j:= 1 TO 6 DO
					PosicionDisponible_aux := 1;
					FOR m:= 0 TO 17 DO
						IF PosicionPiezaAlmacenada[m] = j THEN
							PosicionDisponible_aux := 0;
							EXIT;
						END_IF
					END_FOR
					IF PosicionDisponible_aux = 1 THEN
						PosicionDisponible := j;
						EXIT;
					END_IF
				END_FOR
			ELSIF ((RecogidaPieza.ColorPieza = 2 AND ColorPiezaDescargada[k] = 0) OR ColorPiezaDescargada[k] = 2) AND ContadorPlateado < 6 THEN
				FOR j:= 7 TO 12 DO
					PosicionDisponible_aux := 1;
					FOR m:= 0 TO 17 DO
						IF PosicionPiezaAlmacenada[m] = j THEN
							PosicionDisponible_aux := 0;
							EXIT;
						END_IF
					END_FOR
					IF PosicionDisponible_aux = 1 THEN
						PosicionDisponible := j;
						EXIT;
					END_IF
				END_FOR
			ELSIF ((RecogidaPieza.ColorPieza = 3 AND ColorPiezaDescargada[k] = 0) OR ColorPiezaDescargada[k] = 3) AND ContadorRojo < 6 THEN
				FOR j:= 13 TO 18 DO
					PosicionDisponible_aux := 1;
					FOR m:= 0 TO 17 DO
						IF PosicionPiezaAlmacenada[m] = j THEN
							PosicionDisponible_aux := 0;
							EXIT;
						END_IF
					END_FOR
					IF PosicionDisponible_aux = 1 THEN
						PosicionDisponible := j;
						EXIT;
					END_IF
				END_FOR
			END_IF
			n := 0; 
			WHILE ColorPiezaAlmacenada[n] <> 0 DO
				n := n + 1;
			END_WHILE
		ELSE
			(*Llena el almacén independientemente del color*)
			n := 0;
			PosicionDisponible := 1;
			WHILE ColorPiezaAlmacenada[n] <> 0 DO
				n := n + 1;
				PosicionDisponible := PosicionDisponible + 1;
			END_WHILE
		END_IF
	END_IF
END_IF

(*Guardar fecha, color y posición de la pieza almacenada*) 
IF TrasladoPieza.Estado = Etapas_TrasladoPieza.RecogerCilindro THEN
	PosicionPiezaAlmacenada[n] := PosicionDisponible;
	
	IF ColorPiezaDescargada[k] = 0 THEN
		ColorPiezaAlmacenada[n] := RecogidaPieza.ColorPieza;
	ELSE
		ColorPiezaAlmacenada[n] := ColorPiezaDescargada[k];
	END_IF
	
	IF FechaPiezaDescargada[k] = 0 THEN
		FechaPiezaAlmacenada[n] := RecogidaPieza.Fecha;
	ELSE
		FechaPiezaAlmacenada[n] := getRTC();
	END_IF	
END_IF

(*Contador piezas almacenadas*)
IF TrasladoPieza.Estado = Etapas_TrasladoPieza.Fin THEN	
		IF ColorPiezaAlmacenada[n] = 1 THEN
			ContadorNegro := ContadorNegro + 1;
		ELSIF ColorPiezaAlmacenada[n] = 2 THEN
			ContadorPlateado := ContadorPlateado + 1;
		ELSIF ColorPiezaAlmacenada[n] = 3 THEN 
			ContadorRojo := ContadorRojo + 1;
		END_IF	
END_IF
ContadorTotal := ContadorRojo + ContadorNegro + ContadorPlateado;

(*Posición de la pieza a descargar*)
IF ExtraerPieza.Estado = Etapas_ExtraerPieza.RecogerCilindro1 THEN
	(*MODO AUTOMÁTICO*)
	IF Mando.Estado = Etapas_Mando.F1 OR Mando.Estado = Etapas_Mando.F6 OR Mando.Estado = Etapas_Mando.A2 THEN
		IF Funcionamiento.ModoDescarga = 1 THEN 
			(*Descarga todo el almacén por orden de almacenamiento*)
			FechaReferencia := getRTC(); 
			FOR i := 0 TO 17 DO
				IF FechaPiezaAlmacenada[i] <> 0 AND FechaPiezaAlmacenada[i] < FechaReferencia THEN
					FechaReferencia := FechaPiezaAlmacenada[i];
					k := i;
				END_IF
			END_FOR
			PosicionDescarga := PosicionPiezaAlmacenada[k];
		ELSIF Funcionamiento.ModoDescarga = 2 THEN
			(*Descarga todas las piezas del color seleccionado por orden de almacenamiento*)
			FechaReferencia := getRTC(); 
			IF Funcionamiento.DescargaColor = 1 THEN
				FOR i := 0 TO 17 DO
					IF ColorPiezaAlmacenada[i] = 1 AND FechaPiezaAlmacenada[i] < FechaReferencia THEN
						FechaReferencia := FechaPiezaAlmacenada[i];
						k := i;
					END_IF
				END_FOR
				PosicionDescarga := PosicionPiezaAlmacenada[k];
			ELSIF Funcionamiento.DescargaColor = 2 THEN	
				FOR i := 0 TO 17 DO
					IF ColorPiezaAlmacenada[i] = 2 AND FechaPiezaAlmacenada[i] < FechaReferencia THEN
						FechaReferencia := FechaPiezaAlmacenada[i];
						k := i;
					END_IF
				END_FOR
				PosicionDescarga := PosicionPiezaAlmacenada[k];
			ELSIF Funcionamiento.DescargaColor = 3 THEN	
				FOR i := 0 TO 17 DO
					IF ColorPiezaAlmacenada[i] = 3 AND FechaPiezaAlmacenada[i] < FechaReferencia THEN
						FechaReferencia := FechaPiezaAlmacenada[i];
						k := i;
					END_IF
				END_FOR
				PosicionDescarga := PosicionPiezaAlmacenada[k];
			END_IF
		ELSIF Funcionamiento.ModoDescarga = 3 THEN
			(*Descarga un lote de piezas de cada color por orden de almacenamiento*)
			FechaReferencia := getRTC();
			FOR i := 0 TO 17 DO
				IF (ColorPiezaAlmacenada[i] = 1 AND FechaPiezaAlmacenada[i] < FechaReferencia AND Funcionamiento.NegrasPedidas > 0) 
					OR (ColorPiezaAlmacenada[i] = 2 AND FechaPiezaAlmacenada[i] < FechaReferencia AND Funcionamiento.PlateadasPedidas > 0)
					OR (ColorPiezaAlmacenada[i] = 3 AND FechaPiezaAlmacenada[i] < FechaReferencia AND Funcionamiento.RojasPedidas > 0) THEN
						FechaReferencia := FechaPiezaAlmacenada[i];
						k := i;
				END_IF
			END_FOR
			PosicionDescarga := PosicionPiezaAlmacenada[k];
			IF ColorPiezaAlmacenada[k] = 1  THEN
				Funcionamiento.NegrasPedidas := Funcionamiento.NegrasPedidas - 1;				
			ELSIF ColorPiezaAlmacenada[k] = 2  THEN
				Funcionamiento.PlateadasPedidas := Funcionamiento.PlateadasPedidas - 1;
			ELSIF ColorPiezaAlmacenada[k] = 3  THEN
				Funcionamiento.RojasPedidas := Funcionamiento.RojasPedidas - 1;
			END_IF			
		END_IF
	END_IF 
	
	(*MODO MANUAL*)
	IF Mando.Estado = Etapas_Mando.F4 THEN
		(*Descarga la pieza más antigua del almacén del color escogido por el usuario*)
		FechaReferencia := getRTC(); 
		IF Main.VSO_ColorDescarga = 1 THEN
			FOR i := 0 TO 17 DO
				IF ColorPiezaAlmacenada[i] = 1 AND FechaPiezaAlmacenada[i] < FechaReferencia THEN
					FechaReferencia := FechaPiezaAlmacenada[i];
					k := i;
				END_IF
			END_FOR
			PosicionDescarga := PosicionPiezaAlmacenada[k];
		ELSIF Main.VSO_ColorDescarga = 2 THEN
			FOR i := 0 TO 17 DO
				IF ColorPiezaAlmacenada[i] = 2 AND FechaPiezaAlmacenada[i] < FechaReferencia THEN
					FechaReferencia := FechaPiezaAlmacenada[i];
					k := i;
				END_IF
			END_FOR
			PosicionDescarga := PosicionPiezaAlmacenada[k];
		ELSIF Main.VSO_ColorDescarga = 3 THEN
			FOR i := 0 TO 17 DO
				IF ColorPiezaAlmacenada[i] = 3 AND FechaPiezaAlmacenada[i] < FechaReferencia THEN
					FechaReferencia := FechaPiezaAlmacenada[i];
					k := i;
				END_IF
			END_FOR
			PosicionDescarga := PosicionPiezaAlmacenada[k];
		END_IF
	END_IF
END_IF

(*Borra la pieza extraída del almacén y reduce el contador*)
IF ExtraerPieza.Estado = Etapas_ExtraerPieza.Espera THEN
	IF ColorPiezaAlmacenada[k] = 1 AND ContadorNegro > 0 THEN
		ColorPiezaDescargada[k] := 1;
		ContadorNegro := ContadorNegro - 1;
	ELSIF ColorPiezaAlmacenada[k] = 2 AND ContadorPlateado > 0 THEN
		ColorPiezaDescargada[k] := 2;
		ContadorPlateado := ContadorPlateado - 1;
	ELSIF ColorPiezaAlmacenada[k] = 3 AND ContadorRojo > 0 THEN
		ColorPiezaDescargada[k] := 3; 
		ContadorRojo := ContadorRojo - 1;
	END_IF
	ColorPiezaAlmacenada[k] := 0;	
	FechaPiezaDescargada[k] := FechaPiezaAlmacenada[k];
	FechaPiezaAlmacenada[k] := 0;
	PosicionPiezaAlmacenada[k] := 0;	
END_IF

(*Borra el color y la fecha de la pieza descargada*)
IF SalidaPieza.Estado = Etapas_SalidaPieza.Fin OR TrasladoPieza.Estado = Etapas_TrasladoPieza.Fin THEN
	ColorPiezaDescargada[k] := 0;	
	FechaPiezaDescargada[k] := 0;
END_IF

(*Borra los lotes de piezas pedidas para descargar*)
IF Funcionamiento.BorrarLotes THEN
	Funcionamiento.NegrasPedidas := 0;
	Funcionamiento.PlateadasPedidas := 0;
	Funcionamiento.RojasPedidas := 0;
END_IF

END_PROGRAM

// MyController/Application/ExtraerPieza
PROGRAM ExtraerPieza
VAR_INPUT
	Estado: Etapas_ExtraerPieza;
END_VAR

(*MÁQUINA DE ESTADOS PARA LA DESCARGA DE UNA PIEZA DEL ALMACÉN*)

CASE Estado OF
	
	Etapas_ExtraerPieza.EInicial:
	(*Transición*)
	IF Inicio_ExtraerPieza THEN
		Estado := Etapas_ExtraerPieza.RecogerCilindro1;
	END_IF
	
	Etapas_ExtraerPieza.RecogerCilindro1:
	(*Recoger el cilindro*)
	(*Transición*)
	IF GVL.IN_FC_CilindroAtras THEN
		Estado := Etapas_ExtraerPieza.MoverRobot;
	END_IF
	
	Etapas_ExtraerPieza.MoverRobot:
	(*Mover el robot a la posición del almacén*)
	(*Transición*)
	IF MovimientoRobot.Estado = Etapas_MovimientoRobot.Fin THEN
		Estado := Etapas_ExtraerPieza.AccionarCilindro;
	END_IF
	
	Etapas_ExtraerPieza.AccionarCilindro:
	(*Accionar el cilindro*)
	(*Transición*)
	IF GVL.IN_FC_CilindroDelante THEN
		Estado := Etapas_ExtraerPieza.BajarRobot;
	END_IF
	
	Etapas_ExtraerPieza.BajarRobot:
	(*Bajar el robot una posición*)
	(*Transición*)
	IF MovimientoRobot.Estado = Etapas_MovimientoRobot.Fin THEN
		Estado := Etapas_ExtraerPieza.CerrarPinza;
	END_IF
	
	Etapas_ExtraerPieza.CerrarPinza:
	(*Cerrar la pinza*)
		Estado := Etapas_ExtraerPieza.SubirRobot;
	
	Etapas_ExtraerPieza.SubirRobot:
	(*Subir el robot una posición*)
	(*Transición*)
	IF MovimientoRobot.Estado = Etapas_MovimientoRobot.Fin THEN
		Estado := Etapas_ExtraerPieza.RecogerCilindro2;
	END_IF
	
	Etapas_ExtraerPieza.RecogerCilindro2:
	(*Recoger el cilindro*)
	(*Transición*)
	IF GVL.IN_FC_CilindroAtras THEN
		Estado := Etapas_ExtraerPieza.Espera;
	END_IF
	
	Etapas_ExtraerPieza.Espera:
	(*Final de la extracción, espera para el traslado a la salida*)
		Estado := Etapas_ExtraerPieza.EInicial;

END_CASE

TRANSITION Inicio_ExtraerPieza:
IF Funcionamiento.Estado = Etapas_Funcionamiento.ExtraePieza OR MarchaVSO.Estado = Etapas_MarchaVSO.ExtraePieza THEN
	Inicio_ExtraerPieza := 1;
ELSE
	Inicio_ExtraerPieza := 0;
END_IF
END_TRANSITION

END_PROGRAM

// MyController/Application/MarchaVSO
PROGRAM MarchaVSO
VAR_INPUT
	Estado: Etapas_MarchaVSO;
END_VAR
VAR
	CargaDisponible: BOOL;
	DescargaDisponible: BOOL;
END_VAR

(*MÁQUINA DE ESTADOS DE LA MARCHA DE VERIFICACIÓN SIN ORDEN*)

CASE Estado OF
	
	Etapas_MarchaVSO.EInicial:
	(*Transición*)
	IF Mando.Estado = Etapas_Mando.F4 THEN
		Estado := Etapas_MarchaVSO.Funcionamiento;
	END_IF
	
	Etapas_MarchaVSO.Funcionamiento:
	(*Se selecciona manualmente si hay que cargar una pieza, trasladarla al almacén, extraerla del almacén, llevarla a la salida o no hacer nada*)
	(*Transiciones*)
	IF Recoger THEN 
		Estado := Etapas_MarchaVSO.RecogePieza;
	ELSIF Trasladar THEN
		Estado := Etapas_MarchaVSO.TrasladoPieza;
	ELSIF Extraer THEN
		Estado := Etapas_MarchaVSO.ExtraePieza;
	ELSIF Salir THEN
		Estado := Etapas_MarchaVSO.SalidaPieza;
	ELSIF Finalizar THEN
		Estado := Etapas_MarchaVSO.Fin;
	END_IF
	
	Etapas_MarchaVSO.RecogePieza:
	(*Se recoge una pieza en la entrada*)
	(*Transición*)
	IF RecogidaPieza.Estado = Etapas_RecogidaPieza.Espera THEN
		Estado := Etapas_MarchaVSO.Funcionamiento;
	END_IF
	
	Etapas_MarchaVSO.TrasladoPieza:
	(*Se traslada la pieza al almacén*)
	(*Transición*)
	IF TrasladoPieza.Estado = Etapas_TrasladoPieza.Fin THEN
		Estado := Etapas_MarchaVSO.Espera;
	END_IF
	
	Etapas_MarchaVSO.ExtraePieza:
	(*Se extrae una pieza del almacén*)
	(*Transición*)
	IF ExtraerPieza.Estado = Etapas_ExtraerPieza.Espera THEN
		Estado := Etapas_MarchaVSO.Funcionamiento;
	END_IF
	
	Etapas_MarchaVSO.SalidaPieza:
	(*Se lleva la pieza a la salida*)
	(*Transición*)
	IF SalidaPieza.Estado = Etapas_SalidaPieza.Fin THEN
		Estado := Etapas_MarchaVSO.Espera;
	END_IF
	
	Etapas_MarchaVSO.Espera:
	(*Se comprueba si se continúa en modo manual o cambia al modo automático o se solicitó el test*)
	(*Transición*)
	IF GVL.IN_Aut_Man THEN
		Estado := Etapas_MarchaVSO.Funcionamiento;
	ELSIF NOT GVL.IN_Aut_Man OR Mando.Test THEN
		Estado := Etapas_MarchaVSO.Fin;
	END_IF
	
	Etapas_MarchaVSO.Fin:
		Estado := Etapas_MarchaVSO.EInicial;
	

END_CASE

TRANSITION Recoger:
(*Para que recoja una pieza en la entrada tienen que estar las pinzas abiertas*)
Recoger := NOT GVL.OUT_Pinza AND Main.VSO_Recoger AND GVL.BIT_PiezaEntrada;
END_TRANSITION

TRANSITION Trasladar:
(*Para trasladar la pieza al almacén tiene que haber espacio disponible y las pinzas tienen que estar cerradas*)
IF Funcionamiento.CargaPorColor = 1 THEN
	IF RecogidaPieza.ColorPieza = 1 AND GestionPiezas.ContadorNegro < 6 THEN
		CargaDisponible := 1;
	ELSIF RecogidaPieza.ColorPieza = 2 AND GestionPiezas.ContadorPlateado < 6 THEN
		CargaDisponible := 1;
	ELSIF RecogidaPieza.ColorPieza = 3 AND GestionPiezas.ContadorRojo < 6 THEN
		CargaDisponible := 1;
	ELSE
		CargaDisponible := 0;
	END_IF
ELSE
	CargaDisponible := GestionPiezas.ContadorTotal < 18;
END_IF

Trasladar := CargaDisponible and GVL.OUT_Pinza and Main.VSO_Trasladar;
END_TRANSITION

TRANSITION Extraer:
(*Para extraer una pieza del almacén tienen que estar las pinzas abiertas y haber alguna pieza almacenada del color seleccionado*)
IF (Main.VSO_ColorDescarga = 1 AND GestionPiezas.ContadorNegro > 0) OR (Main.VSO_ColorDescarga = 2 AND 
	GestionPiezas.ContadorPlateado > 0) OR (Main.VSO_ColorDescarga = 3 AND GestionPiezas.ContadorRojo > 0) THEN
	DescargaDisponible := 1;
ELSE
	DescargaDisponible := 0;
END_IF

Extraer := DescargaDisponible AND NOT GVL.OUT_Pinza AND Main.VSO_Extraer;
END_TRANSITION

TRANSITION Salir:
(*Para llevar una pieza a la salida tienen que estar las pinzas cerradas*)
Salir := GVL.OUT_Pinza and Main.VSO_Salir;
END_TRANSITION

TRANSITION Finalizar:
Finalizar := Main.VSO_Nada and NOT GVL.OUT_Pinza;
END_TRANSITION

END_PROGRAM

// MyController/Application/SalidaPieza
PROGRAM SalidaPieza
VAR_INPUT
	Estado: Etapas_SalidaPieza;
END_VAR

(*MÁQUINA DE ESTADOS PARA EL TRASLADO DE LA PIEZA A LA SALIDA*)

CASE Estado OF
	
	Etapas_SalidaPieza.EInicial:
	(*Transición*)
	IF Inicio_SalidaPieza THEN
		Estado := Etapas_SalidaPieza.MoverRobot;
	END_IF
	
	Etapas_SalidaPieza.MoverRobot:
	(*Mover el robot a la posición de salida*)
	(*Transición*)
	IF MovimientoRobot.Estado = Etapas_MovimientoRobot.Fin THEN
		Estado := Etapas_SalidaPieza.AccionarCilindro;
	END_IF
	
	Etapas_SalidaPieza.AccionarCilindro:
	(*Accionar el cilindro*)
	(*Transición*)
	IF GVL.IN_FC_CilindroDelante THEN
		Estado := Etapas_SalidaPieza.AbrirPinza;
	END_IF
	
	Etapas_SalidaPieza.AbrirPinza:
	(*Abrir la pinza*)
		Estado := Etapas_SalidaPieza.SubirRobot;
		
	Etapas_SalidaPieza.SubirRobot:
	(*Subir el robot una posición*)
	(*Transición*)
	IF MovimientoRobot.Estado = Etapas_MovimientoRobot.Fin THEN
		Estado := Etapas_SalidaPieza.RecogerCilindro;
	END_IF
	
	Etapas_SalidaPieza.RecogerCilindro:
	(*Recoger el cilindro*)
	(*Transición*)
	IF GVL.IN_FC_CilindroAtras THEN
		Estado := Etapas_SalidaPieza.Fin;
	END_IF
	
	
	Etapas_SalidaPieza.Fin:
	(*Final de la salida de la pieza*)
		Estado := Etapas_SalidaPieza.EInicial;	

END_CASE

TRANSITION Inicio_SalidaPieza:
IF Funcionamiento.Estado = Etapas_Funcionamiento.SalidaPieza OR Funcionamiento.Estado = Etapas_Funcionamiento.SalidaPieza2
	OR MarchaVSO.Estado = Etapas_MarchaVSO.SalidaPieza THEN
	Inicio_SalidaPieza := 1;
ELSE
	Inicio_SalidaPieza := 0;
END_IF
END_TRANSITION

END_PROGRAM

// MyController/Application/Inicializacion
PROGRAM Inicializacion
VAR_INPUT
	Estado: Etapas_Inicializacion;
END_VAR

(*MÁQUINA DE ESTADOS PARA LA INICIALIZACIÓN*)
CASE Estado OF
	
	Etapas_Inicializacion.EInicial:
	(*Transición*)
	IF Mando.Estado = Etapas_Mando.A6 THEN
		Estado := Etapas_Inicializacion.Espera;
	END_IF
	
	Etapas_Inicializacion.Espera:
	(*Se recoge el cilindro y se abre la pinza*)
	(*Transición*)
	IF GVL.IN_Reset OR Control.HMI_Reset THEN
		Estado := Etapas_Inicializacion.MoverRobot;
	END_IF
	
	Etapas_Inicializacion.MoverRobot:
	(*Mover robot a la posición de referencia*)
	(*Transición*)
	IF MovimientoRobot.Estado = Etapas_MovimientoRobot.Fin  THEN
		Estado := Etapas_Inicializacion.Fin;
	END_IF
			
	Etapas_Inicializacion.Fin:
	(*Final de la inicialización*)
		Estado := Etapas_Inicializacion.EInicial;

END_CASE

END_PROGRAM

// MyController/Application/PosicionRobot
PROGRAM PosicionRobot
VAR
	CoordenadaH: INT;
	CoordenadaV: INT;
	Posicion: INT;
	i: INT;
	EnviarCoordenadas: INT;
END_VAR

(*Posición*)
IF TrasladoPieza.Estado = Etapas_TrasladoPieza.MoverRobot THEN
	Posicion := GestionPiezas.PosicionDisponible;
ELSIF ExtraerPieza.Estado = Etapas_ExtraerPieza.MoverRobot THEN
	Posicion := GestionPiezas.PosicionDescarga;
ELSIF Inicializacion.Estado = Etapas_Inicializacion.MoverRobot THEN
	Posicion := 0; (*Referencia*)
ELSIF RecogidaPieza.Estado = Etapas_RecogidaPieza.MoverRobot THEN
	Posicion := 19; (*Receptor de pieza e identificador de color*)
ELSIF SalidaPieza.Estado = Etapas_SalidaPieza.MoverRobot OR Test.Estado = Etapas_Test.MoverRobot THEN
	Posicion := 20; (*Descarga de pieza*)	
END_IF


(*Coordenadas de las distintas posiciones*)
IF Funcionamiento.CargaPorColor = 1 THEN
	(*Posicionamiento de piezas dependiendo del color: Nivel 1 - negro, Nivel 2 - plateado, Nivel 3 - rojo*)
	CASE Posicion OF
	0: CoordenadaV:=0; CoordenadaH:= 7; (*Referencia*)
	1: CoordenadaV:=1; CoordenadaH:=5; (*Nivel 1, posición F*)
	2: CoordenadaV:=1; CoordenadaH:=4; (*Nivel 1, posición E*)
	3: CoordenadaV:=1; CoordenadaH:=3; (*Nivel 1, posición D*)
	4: CoordenadaV:=1; CoordenadaH:=2; (*Nivel 1, posición C*)
	5: CoordenadaV:=1; CoordenadaH:=1; (*Nivel 1, posición B*)
	6: CoordenadaV:=1; CoordenadaH:=0; (*Nivel 1, posición A*)
	7: CoordenadaV:=3; CoordenadaH:=5; (*Nivel 2, posición F*)
	8: CoordenadaV:=3; CoordenadaH:=4; (*Nivel 2, posición E*)
	9: CoordenadaV:=3; CoordenadaH:=3; (*Nivel 2, posición D*)
	10: CoordenadaV:=3; CoordenadaH:=2; (*Nivel 2, posición C*)
	11: CoordenadaV:=3; CoordenadaH:=1; (*Nivel 2, posición B*)
	12: CoordenadaV:=3; CoordenadaH:=0; (*Nivel 2, posición A*)
	13: CoordenadaV:=6; CoordenadaH:=5; (*Nivel 3, posición F*)
	14: CoordenadaV:=6; CoordenadaH:=4; (*Nivel 3, posición E*)
	15: CoordenadaV:=6; CoordenadaH:=3; (*Nivel 3, posición D*)
	16: CoordenadaV:=6; CoordenadaH:=2; (*Nivel 3, posición C*)
	17: CoordenadaV:=6; CoordenadaH:=1; (*Nivel 3, posición B*)
	18: CoordenadaV:=6; CoordenadaH:=0; (*Nivel 3, posición A*)
	19: CoordenadaV:=5; CoordenadaH:=6; (*Receptor de pieza e identificador de color*)
	20: CoordenadaV:=7; CoordenadaH:=7; (*Descarga de pieza*)
	END_CASE
ELSE
	(*Posicionamiento de piezas independientemente del color*)
	CASE Posicion OF
	0: CoordenadaV:=0; CoordenadaH:= 7; (*Referencia*)
	1: CoordenadaV:=1; CoordenadaH:=5; (*Nivel 1, posición F*)
	2: CoordenadaV:=3; CoordenadaH:=5; (*Nivel 2, posición F*)
	3: CoordenadaV:=6; CoordenadaH:=5; (*Nivel 3, posición F*)
	4: CoordenadaV:=1; CoordenadaH:=4; (*Nivel 1, posición E*)
	5: CoordenadaV:=3; CoordenadaH:=4; (*Nivel 2, posición E*)
	6: CoordenadaV:=6; CoordenadaH:=4; (*Nivel 3, posición E*)
	7: CoordenadaV:=1; CoordenadaH:=3; (*Nivel 1, posición D*)
	8: CoordenadaV:=3; CoordenadaH:=3; (*Nivel 2, posición D*)
	9: CoordenadaV:=6; CoordenadaH:=3; (*Nivel 3, posición D*)
	10: CoordenadaV:=1; CoordenadaH:=2; (*Nivel 1, posición C*)
	11: CoordenadaV:=3; CoordenadaH:=2; (*Nivel 2, posición C*)
	12: CoordenadaV:=6; CoordenadaH:=2; (*Nivel 3, posición C*)
	13: CoordenadaV:=1; CoordenadaH:=1; (*Nivel 1, posición B*)
	14: CoordenadaV:=3; CoordenadaH:=1; (*Nivel 2, posición B*)
	15: CoordenadaV:=6; CoordenadaH:=1; (*Nivel 3, posición B*)
	16: CoordenadaV:=1; CoordenadaH:=0; (*Nivel 1, posición A*)
	17: CoordenadaV:=3; CoordenadaH:=0; (*Nivel 2, posición A*)
	18: CoordenadaV:=6; CoordenadaH:=0; (*Nivel 3, posición A*)
	19: CoordenadaV:=5; CoordenadaH:=6; (*Receptor de pieza e identificador de color*)
	20: CoordenadaV:=7; CoordenadaH:=7; (*Descarga de pieza*)
	END_CASE
END_IF

(*Bajar robot en la posición*)
IF RecogidaPieza.Estado = Etapas_RecogidaPieza.BajarRobot THEN
	CoordenadaV := CoordenadaV + 2;
ELSIF TrasladoPieza.Estado = Etapas_TrasladoPieza.BajarRobot OR ExtraerPieza.Estado = Etapas_ExtraerPieza.BajarRobot THEN
	CoordenadaV := CoordenadaV + 1;
ELSIF Test.Estado = Etapas_Test.BajarRobot THEN
	CoordenadaV := 7;
END_IF

(*Subir robot en la posición*)
IF RecogidaPieza.Estado = Etapas_RecogidaPieza.CerrarPinza THEN
	CoordenadaV := CoordenadaV - 2;
ELSIF TrasladoPieza.Estado = Etapas_TrasladoPieza.AbrirPinza OR ExtraerPieza.Estado = Etapas_ExtraerPieza.CerrarPinza OR 
		SalidaPieza.Estado = Etapas_SalidaPieza.SubirRobot THEN
	CoordenadaV := CoordenadaV - 1;
ELSIF Test.Estado = Etapas_Test.SubirRobot THEN
	CoordenadaV := 0;
END_IF

(*Enviar coordenadas*)
IF MovimientoRobot.Estado = Etapas_MovimientoRobot.EnvioHorizontal THEN
	EnviarCoordenadas := CoordenadaH;	
END_IF
IF MovimientoRobot.Estado = Etapas_MovimientoRobot.EnvioVertical THEN
	EnviarCoordenadas := CoordenadaV;
END_IF

END_PROGRAM

// MyController/Application/Pantalla
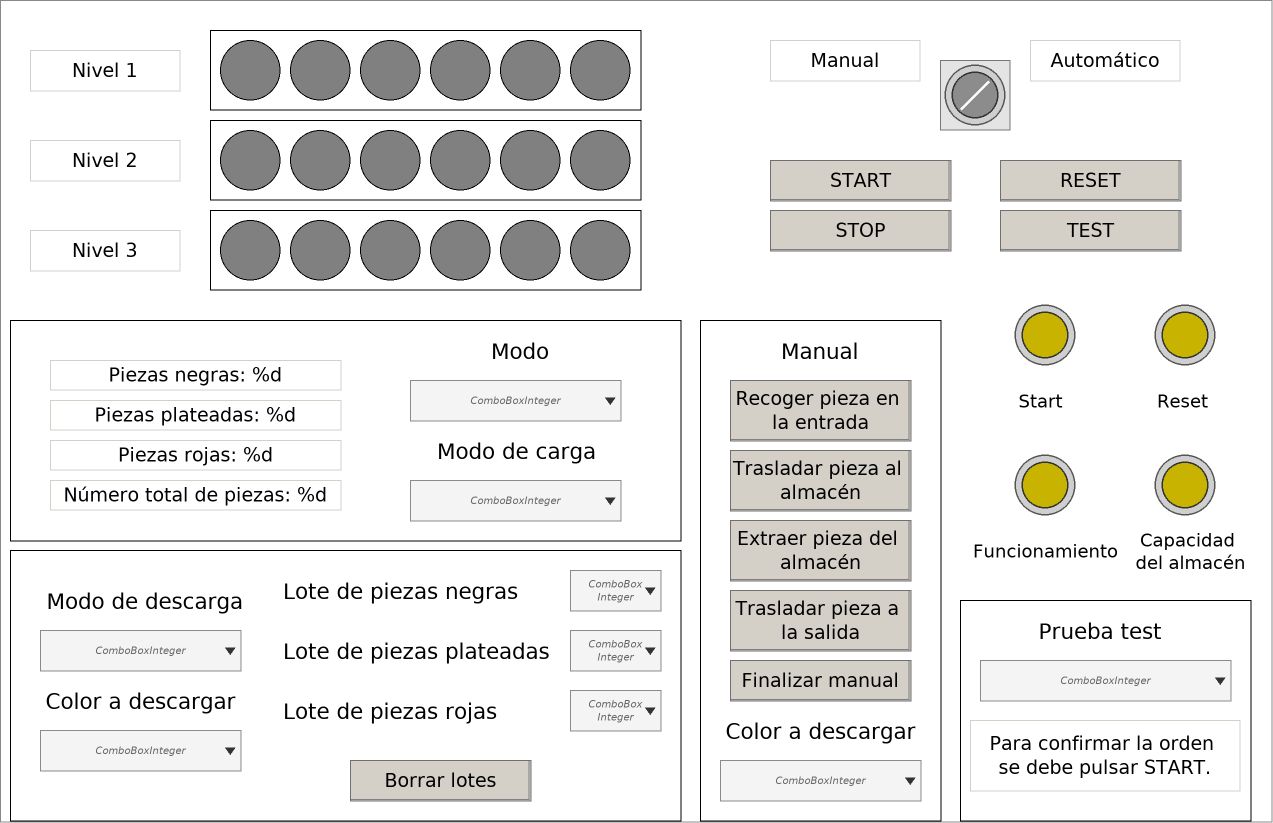
VISUALIZATION Pantalla  // 1273x823
    RoundedRectangle (10,320 671x221)
    RoundedRectangle (700,320 241x501), invisible if: Control.InvManual
    RoundedRectangle (960,600 291x221), invisible if: Control.InvTest
    RoundedRectangle (10,550 671x271), invisible if: Control.InvDescarga
    RoundedRectangle (210,210 431x80)
    Ellipse (570,220 60x60), colour toggle: Control.PiezaNegra18, invisible if: Control.InvNegra18
    Ellipse (500,220 60x60), colour toggle: Control.PiezaNegra15, invisible if: Control.InvNegra15
    Ellipse (430,220 60x60), colour toggle: Control.PiezaNegra12, invisible if: Control.InvNegra12
    Ellipse (360,220 60x60), colour toggle: Control.PiezaNegra9, invisible if: Control.InvNegra9
    Ellipse (290,220 60x60), colour toggle: Control.PiezaNegra6, invisible if: Control.InvNegra6
    Ellipse (220,220 60x60), colour toggle: Control.PiezaNegra3, invisible if: Control.InvNegra3
    RoundedRectangle (210,120 431x80)
    Ellipse (570,130 60x60), colour toggle: Control.PiezaNegra17, invisible if: Control.InvNegra17
    Ellipse (500,130 60x60), colour toggle: Control.PiezaNegra14, invisible if: Control.InvNegra14
    Ellipse (430,130 60x60), colour toggle: Control.PiezaNegra11, invisible if: Control.InvNegra11
    Ellipse (360,130 60x60), colour toggle: Control.PiezaNegra8, invisible if: Control.InvNegra8
    Ellipse (290,130 60x60), colour toggle: Control.PiezaNegra5, invisible if: Control.InvNegra5
    Ellipse (220,130 60x60), colour toggle: Control.PiezaNegra2, invisible if: Control.InvNegra2
    RoundedRectangle (210,30 431x80)
    Ellipse (570,40 60x60), colour toggle: Control.PiezaNegra16, invisible if: Control.InvNegra16
    Ellipse (500,40 60x60), colour toggle: Control.PiezaNegra13, invisible if: Control.InvNegra13
    Ellipse (430,40 60x60), colour toggle: Control.PiezaNegra10, invisible if: Control.InvNegra10
    Ellipse (360,40 60x60), colour toggle: Control.PiezaNegra7, invisible if: Control.InvNegra7
    Ellipse (290,40 60x60), colour toggle: Control.PiezaNegra4, invisible if: Control.InvNegra4
    Ellipse (220,40 60x60)
    Ellipse (220,40 60x60), colour toggle: Control.PiezaNegra1, invisible if: Control.InvNegra1
    Ellipse (220,40 60x60), colour toggle: Control.PiezaPlateadaRoja1, invisible if: Control.InvPlateadaRoja1
    Textfield (30,50 150x41), "Nivel 1"
    Textfield (30,140 150x41), "Nivel 2"
    Textfield (30,230 150x41), "Nivel 3"
    Lamp1 (1010,300 70x70), variable: GVL.OUT_Piloto_Start, style: Lamp-Lamp1-Yellow
    Lamp1 (1150,300 70x70), variable: GVL.OUT_Piloto_Reset, style: Lamp-Lamp1-Yellow
    Lamp1 (1010,450 70x70), variable: GVL.OUT_Piloto_Q1, style: Lamp-Lamp1-Yellow
    Lamp1 (1150,450 70x70), variable: GVL.OUT_Piloto_Q2, style: Lamp-Lamp1-Yellow
    Label (970,380 141x43), "Start"
    Label (1112,380 141x43), "Reset"
    Label (960,530 171x43), "Funcionamiento"
    Label (1110,530 161x43), "Capacidad del almacén"
    Button (770,160 181x41), "START"
        tap Control.HMI_Start
    Button (770,210 181x41), "STOP"
        tap Control.HMI_Stop
    Button (1000,160 181x41), "RESET"
        tap Control.HMI_Reset
    Button (1000,210 181x41), "TEST"
        toggle Mando.Test
    RotarySwitch (940,60 70x70), variable: GVL.IN_Aut_Man, behaviour: TOGGLE, style: Switch-RotarySwitch-Gray
    ComboBoxInteger (410,380 211x41), variable: Funcionamiento.ModoFuncionamiento, text list: 'Funcionamiento_Lista'
    Label (460,330 120x43), "Modo"
    ComboBoxInteger (410,480 211x41), variable: Funcionamiento.CargaPorColor, invisible if: Control.InvCarga, input disabled if: Control.BloqueoCargaColor, text list: 'Carga_Lista'
    Label (410,430 213x43), "Modo de carga", invisible if: Control.InvCarga
    ComboBoxInteger (40,630 201x41), variable: Funcionamiento.ModoDescarga, invisible if: Control.InvDescarga, text list: 'Descarga_Lista'
    Label (30,580 230x43), "Modo de descarga", invisible if: Control.InvDescarga
    ComboBoxInteger (40,730 201x41), variable: Funcionamiento.DescargaColor, invisible if: Control.InvDesColor, text list: 'DescargaColor_Lista'
    Label (30,680 221x43), "Color a descargar", invisible if: Control.InvDesColor
    ComboBoxInteger (570,570 91x41), variable: Funcionamiento.NegrasPedidas, invisible if: Control.InvDesLotes
    Label (280,570 270x43), "Lote de piezas negras", invisible if: Control.InvDesLotes
    ComboBoxInteger (570,630 91x41), variable: Funcionamiento.PlateadasPedidas, invisible if: Control.InvDesLotes
    Label (280,630 270x43), "Lote de piezas plateadas", invisible if: Control.InvDesLotes
    ComboBoxInteger (570,690 91x41), variable: Funcionamiento.RojasPedidas, invisible if: Control.InvDesLotes
    Button (350,760 181x41), "Borrar lotes", invisible if: Control.InvDesLotes, input disabled if: Control.BloqueoLotes
        OnMouseDown:  ToggleVariable=Funcionamiento.BorrarLotes
    Label (280,690 270x43), "Lote de piezas rojas", invisible if: Control.InvDesLotes
    ComboBoxInteger (980,660 251x41), variable: Test.ModoTest, invisible if: Control.InvTest, text list: 'Test_Lista'
    Label (1010,610 180x43), "Prueba test", invisible if: Control.InvTest
    Textfield (970,720 270x71), "Para confirmar la orden se debe pulsar START.", invisible if: Control.InvTest
    Textfield (1030,40 150x41), "Automático", colour toggle: Control.ColorAutomatico
    Textfield (770,40 150x41), "Manual", colour toggle: Control.ColorManual
    Textfield (50,360 291x30), "Piezas negras: %d", text variable: GestionPiezas.ContadorNegro
    Textfield (50,400 291x30), "Piezas plateadas: %d", text variable: GestionPiezas.ContadorPlateado
    Textfield (50,440 291x30), "Piezas rojas: %d", text variable: GestionPiezas.ContadorRojo
    Textfield (50,480 291x30), "Número total de piezas: %d", text variable: GestionPiezas.ContadorTotal
    Ellipse (220,130 60x60), colour toggle: Control.PiezaPlateadaRoja2, invisible if: Control.InvPlateadaRoja2
    Ellipse (220,220 60x60), colour toggle: Control.PiezaPlateadaRoja3, invisible if: Control.InvPlateadaRoja3
    Ellipse (290,40 60x60), colour toggle: Control.PiezaPlateadaRoja4, invisible if: Control.InvPlateadaRoja4
    Ellipse (290,130 60x60), colour toggle: Control.PiezaPlateadaRoja5, invisible if: Control.InvPlateadaRoja5
    Ellipse (290,220 60x60), colour toggle: Control.PiezaPlateadaRoja6, invisible if: Control.InvPlateadaRoja6
    Ellipse (360,40 60x60), colour toggle: Control.PiezaPlateadaRoja7, invisible if: Control.InvPlateadaRoja7
    Ellipse (360,130 60x60), colour toggle: Control.PiezaPlateadaRoja8, invisible if: Control.InvPlateadaRoja8
    Ellipse (360,220 60x60), colour toggle: Control.PiezaPlateadaRoja9, invisible if: Control.InvPlateadaRoja9
    Ellipse (430,40 60x60), colour toggle: Control.PiezaPlateadaRoja10, invisible if: Control.InvPlateadaRoja10
    Ellipse (430,130 60x60), colour toggle: Control.PiezaPlateadaRoja11, invisible if: Control.InvPlateadaRoja11
    Ellipse (430,220 60x60), colour toggle: Control.PiezaPlateadaRoja12, invisible if: Control.InvPlateadaRoja12
    Ellipse (500,40 60x60), colour toggle: Control.PiezaPlateadaRoja13, invisible if: Control.InvPlateadaRoja13
    Ellipse (500,130 60x60), colour toggle: Control.PiezaPlateadaRoja14, invisible if: Control.InvPlateadaRoja14
    Ellipse (500,220 60x60), colour toggle: Control.PiezaPlateadaRoja15, invisible if: Control.InvPlateadaRoja15
    Ellipse (570,40 60x60), colour toggle: Control.PiezaPlateadaRoja16, invisible if: Control.InvPlateadaRoja16
    Ellipse (570,130 60x60), colour toggle: Control.PiezaPlateadaRoja17, invisible if: Control.InvPlateadaRoja17
    Ellipse (570,220 60x60), colour toggle: Control.PiezaPlateadaRoja18, invisible if: Control.InvPlateadaRoja18
    Button (730,380 181x61), "Recoger pieza en la entrada", invisible if: Control.InvManual, input disabled if: Control.BloqueoManPinzaCerrada
        tap Main.VSO_Recoger
    Button (730,450 181x61), "Trasladar pieza al almacén", invisible if: Control.InvManual, input disabled if: Control.BloqueoManPinzaAbierta
        tap Main.VSO_Trasladar
    Button (730,520 181x61), "Extraer pieza del almacén", invisible if: Control.InvManual, input disabled if: Control.BloqueoManPinzaCerrada
        tap Main.VSO_Extraer
    Button (730,590 181x61), "Trasladar pieza a la salida", invisible if: Control.InvManual, input disabled if: Control.BloqueoManPinzaAbierta
        tap Main.VSO_Salir
    Button (730,660 181x41), "Finalizar manual", invisible if: Control.InvManual, input disabled if: Control.BloqueoManPinzaCerrada
        tap Main.VSO_Nada
    Label (730,330 180x43), "Manual", invisible if: Control.InvManual
    Label (710,710 221x43), "Color a descargar", invisible if: Control.InvManual
    ComboBoxInteger (720,760 201x41), variable: Main.VSO_ColorDescarga, invisible if: Control.InvManual, text list: 'DescargaColor_Lista'
END_VISUALIZATION

(* text list Pantallas_Lista (id | default)
  0 | Pantalla Principal
  1 | Modo Automático
  2 | Modo Manual
  3 | Test
   |  *)

(* text list Funcionamiento_Lista (id | default)
  0 | No seleccionado
  1 | Carga
  2 | Descarga
  3 | No almacena
  4 | Carga y descarga
   |  *)

(* text list Descarga_Lista (id | default)
  0 | No descarga
  1 | Todo el almacén
  2 | Por color
  3 | Por lotes
   |  *)

(* text list DescargaColor_Lista (id | default)
  0 | No seleccionado
  1 | Negro
  2 | Plateado
  3 | Rojo
   |  *)

(* text list Test_Lista (id | default)
  0 | No seleccionado
  1 | Subir robot
  2 | Bajar robot
  3 | Estirar cilindro
  4 | Recoger cilindro
  5 | Abrir pinza
  6 | Cerrar pinza
   |  *)

(* text list Carga_Lista (id | default)
  0 | Carga indiferente
  1 | Carga por color
   |  *)
